REGION Network 158: Lệnh chạy động cơ khuấy Bồn 4 (Coil thường)
   RUNG wire#powerrail
      Contact( "AGTR3263_Should_Run" )
      I_Contact( "PLC2_Loi_Tong" )
      Coil( "AGTR3263_Khuay_Bon4" )
   END_RUNG
   // the same network as SCL:
   "AGTR3263_Khuay_Bon4" := "AGTR3263_Should_Run" AND NOT "PLC2_Loi_Tong";
END_REGION

REGION Network 159: Lệnh đảo chiều động cơ khuấy Bồn 4 (Coil thường)
   RUNG wire#powerrail
      Contact( "PLC2_Step_Bon4_Khuay_Nghich" )
      I_Contact( "PLC2_Loi_Tong" )
      Coil( "AGTR3263_Dao_Chieu" )
   END_RUNG
   // the same network as SCL:
   "AGTR3263_Dao_Chieu" := "PLC2_Step_Bon4_Khuay_Nghich" AND NOT "PLC2_Loi_Tong";
END_REGION

REGION Network 160: Mở van xả đáy Bồn 4 số 1 khi bơm chuyển Nhánh 2 chạy
   RUNG wire#powerrail
      Contact( "Pump3265_Chuyen_Nhanh2" )
      I_Contact( "PLC2_Loi_Tong" )
      Coil( "V3247_Xa_Bon4" )
   END_RUNG
   // the same network as SCL:
   "V3247_Xa_Bon4" := "Pump3265_Chuyen_Nhanh2" AND NOT "PLC2_Loi_Tong";
END_REGION

REGION Network 161: Mở van xả đáy Bồn 4 số 2 khi bơm chuyển Nhánh 2 chạy
   RUNG wire#powerrail
      Contact( "Pump3265_Chuyen_Nhanh2" )
      I_Contact( "PLC2_Loi_Tong" )
      Coil( "V3248_Xa_Bon4" )
   END_RUNG
   // the same network as SCL:
   "V3248_Xa_Bon4" := "Pump3265_Chuyen_Nhanh2" AND NOT "PLC2_Loi_Tong";
END_REGION

REGION Network 162: Mở van xả đáy Bồn 4 số 3 khi bơm chuyển Nhánh 2 chạy
   RUNG wire#powerrail
      Contact( "Pump3265_Chuyen_Nhanh2" )
      I_Contact( "PLC2_Loi_Tong" )
      Coil( "V3249_Xa_Bon4" )
   END_RUNG
   // the same network as SCL:
   "V3249_Xa_Bon4" := "Pump3265_Chuyen_Nhanh2" AND NOT "PLC2_Loi_Tong";
END_REGION

REGION Network 163: Reset CV nước Bồn 3 khi không dosing
   RUNG wire#powerrail
      I_Contact( "PLC2_Step_Bon3_Dosing" )
      { S7_GenerateENO := "TRUE" } Move(in := 0.0, out1 => "CV3211_Nuoc_Bon3")
   END_RUNG
   // the same network as SCL:
   IF NOT "PLC2_Step_Bon3_Dosing" THEN "CV3211_Nuoc_Bon3" := 0.0; END_IF;
END_REGION

REGION Network 164: Reset CV nước Bồn 3 khi Stop hoặc Lỗi tổng PLC2
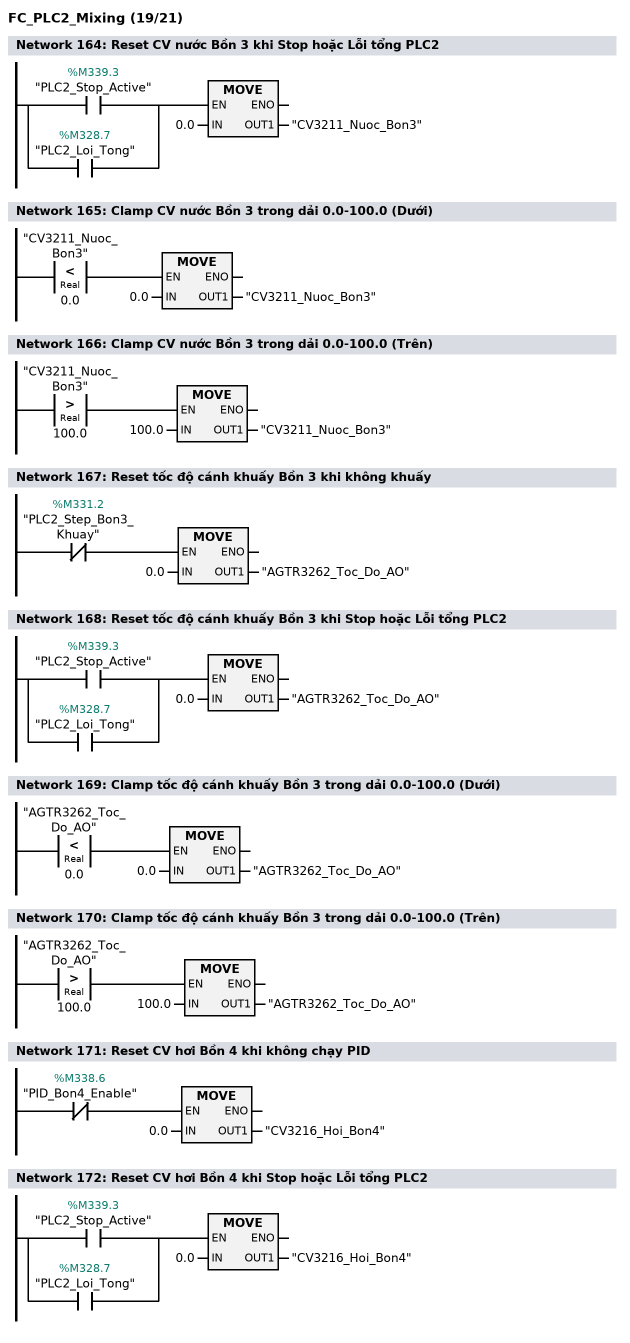
   RUNG wire#powerrail
      Contact( "PLC2_Stop_Active" )
      wire#w1
      { S7_GenerateENO := "TRUE" } Move(in := 0.0, out1 => "CV3211_Nuoc_Bon3")
   END_RUNG
   RUNG wire#powerrail
      Contact( "PLC2_Loi_Tong" )
   END_RUNG wire#w1
   // the same network as SCL:
   IF "PLC2_Stop_Active" OR "PLC2_Loi_Tong" THEN "CV3211_Nuoc_Bon3" := 0.0; END_IF;
END_REGION

REGION Network 165: Clamp CV nước Bồn 3 trong dải 0.0-100.0 (Dưới)
   RUNG wire#powerrail
      { S7_Templates := "SrcType := Real" } LT_Contact(in1 := "CV3211_Nuoc_Bon3", in2 := 0.0)
      { S7_GenerateENO := "TRUE" } Move(in := 0.0, out1 => "CV3211_Nuoc_Bon3")
   END_RUNG
   // the same network as SCL:
   IF "CV3211_Nuoc_Bon3" < 0.0 THEN "CV3211_Nuoc_Bon3" := 0.0; END_IF;
END_REGION

REGION Network 166: Clamp CV nước Bồn 3 trong dải 0.0-100.0 (Trên)
   RUNG wire#powerrail
      { S7_Templates := "SrcType := Real" } GT_Contact(in1 := "CV3211_Nuoc_Bon3", in2 := 100.0)
      { S7_GenerateENO := "TRUE" } Move(in := 100.0, out1 => "CV3211_Nuoc_Bon3")
   END_RUNG
   // the same network as SCL:
   IF "CV3211_Nuoc_Bon3" > 100.0 THEN "CV3211_Nuoc_Bon3" := 100.0; END_IF;
END_REGION

REGION Network 167: Reset tốc độ cánh khuấy Bồn 3 khi không khuấy
   RUNG wire#powerrail
      I_Contact( "PLC2_Step_Bon3_Khuay" )
      { S7_GenerateENO := "TRUE" } Move(in := 0.0, out1 => "AGTR3262_Toc_Do_AO")
   END_RUNG
   // the same network as SCL:
   IF NOT "PLC2_Step_Bon3_Khuay" THEN "AGTR3262_Toc_Do_AO" := 0.0; END_IF;
END_REGION

REGION Network 168: Reset tốc độ cánh khuấy Bồn 3 khi Stop hoặc Lỗi tổng PLC2
   RUNG wire#powerrail
      Contact( "PLC2_Stop_Active" )
      wire#w1
      { S7_GenerateENO := "TRUE" } Move(in := 0.0, out1 => "AGTR3262_Toc_Do_AO")
   END_RUNG
   RUNG wire#powerrail
      Contact( "PLC2_Loi_Tong" )
   END_RUNG wire#w1
   // the same network as SCL:
   IF "PLC2_Stop_Active" OR "PLC2_Loi_Tong" THEN "AGTR3262_Toc_Do_AO" := 0.0; END_IF;
END_REGION

REGION Network 169: Clamp tốc độ cánh khuấy Bồn 3 trong dải 0.0-100.0 (Dưới)
   RUNG wire#powerrail
      { S7_Templates := "SrcType := Real" } LT_Contact(in1 := "AGTR3262_Toc_Do_AO", in2 := 0.0)
      { S7_GenerateENO := "TRUE" } Move(in := 0.0, out1 => "AGTR3262_Toc_Do_AO")
   END_RUNG
   // the same network as SCL:
   IF "AGTR3262_Toc_Do_AO" < 0.0 THEN "AGTR3262_Toc_Do_AO" := 0.0; END_IF;
END_REGION

REGION Network 170: Clamp tốc độ cánh khuấy Bồn 3 trong dải 0.0-100.0 (Trên)
   RUNG wire#powerrail
      { S7_Templates := "SrcType := Real" } GT_Contact(in1 := "AGTR3262_Toc_Do_AO", in2 := 100.0)
      { S7_GenerateENO := "TRUE" } Move(in := 100.0, out1 => "AGTR3262_Toc_Do_AO")
   END_RUNG
   // the same network as SCL:
   IF "AGTR3262_Toc_Do_AO" > 100.0 THEN "AGTR3262_Toc_Do_AO" := 100.0; END_IF;
END_REGION

REGION Network 171: Reset CV hơi Bồn 4 khi không chạy PID
   RUNG wire#powerrail
      I_Contact( "PID_Bon4_Enable" )
      { S7_GenerateENO := "TRUE" } Move(in := 0.0, out1 => "CV3216_Hoi_Bon4")
   END_RUNG
   // the same network as SCL:
   IF NOT "PID_Bon4_Enable" THEN "CV3216_Hoi_Bon4" := 0.0; END_IF;
END_REGION

REGION Network 172: Reset CV hơi Bồn 4 khi Stop hoặc Lỗi tổng PLC2
   RUNG wire#powerrail
      Contact( "PLC2_Stop_Active" )
      wire#w1
      { S7_GenerateENO := "TRUE" } Move(in := 0.0, out1 => "CV3216_Hoi_Bon4")
   END_RUNG
   RUNG wire#powerrail
      Contact( "PLC2_Loi_Tong" )
   END_RUNG wire#w1
   // the same network as SCL:
   IF "PLC2_Stop_Active" OR "PLC2_Loi_Tong" THEN "CV3216_Hoi_Bon4" := 0.0; END_IF;
END_REGION

REGION Network 173: Clamp CV hơi Bồn 4 trong dải 0.0-100.0 (Dưới)
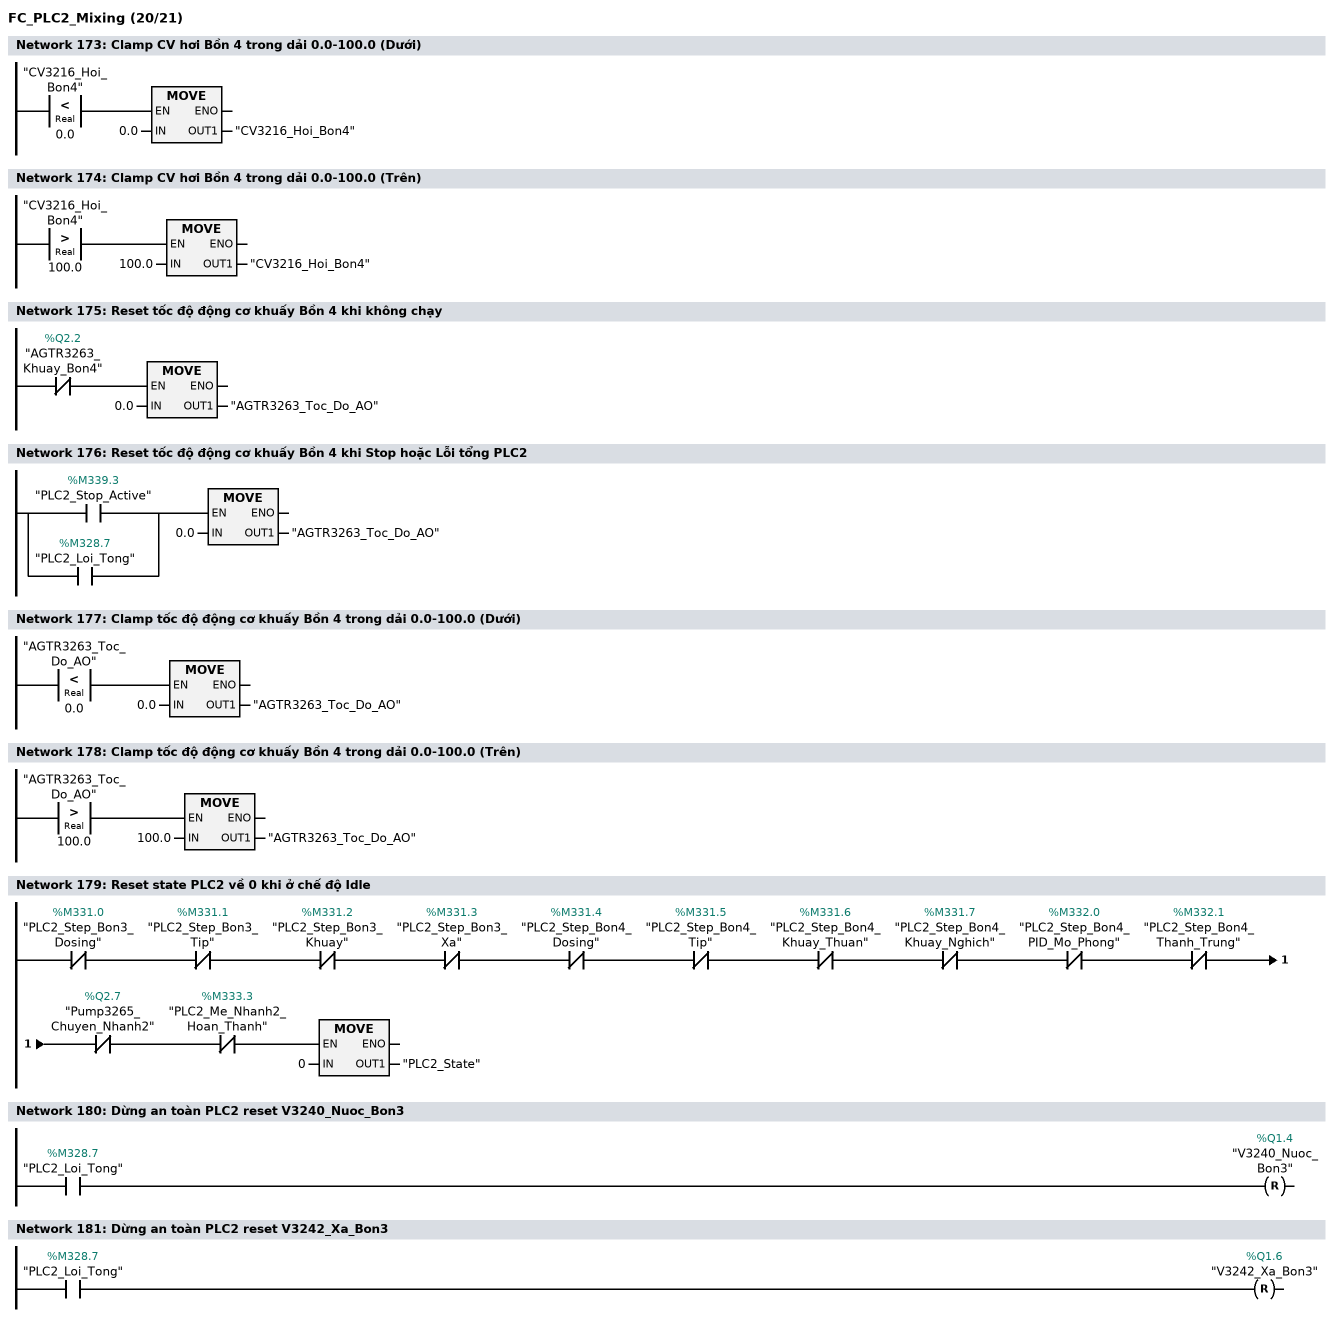
   RUNG wire#powerrail
      { S7_Templates := "SrcType := Real" } LT_Contact(in1 := "CV3216_Hoi_Bon4", in2 := 0.0)
      { S7_GenerateENO := "TRUE" } Move(in := 0.0, out1 => "CV3216_Hoi_Bon4")
   END_RUNG
   // the same network as SCL:
   IF "CV3216_Hoi_Bon4" < 0.0 THEN "CV3216_Hoi_Bon4" := 0.0; END_IF;
END_REGION

REGION Network 174: Clamp CV hơi Bồn 4 trong dải 0.0-100.0 (Trên)
   RUNG wire#powerrail
      { S7_Templates := "SrcType := Real" } GT_Contact(in1 := "CV3216_Hoi_Bon4", in2 := 100.0)
      { S7_GenerateENO := "TRUE" } Move(in := 100.0, out1 => "CV3216_Hoi_Bon4")
   END_RUNG
   // the same network as SCL:
   IF "CV3216_Hoi_Bon4" > 100.0 THEN "CV3216_Hoi_Bon4" := 100.0; END_IF;
END_REGION

REGION Network 175: Reset tốc độ động cơ khuấy Bồn 4 khi không chạy
   RUNG wire#powerrail
      I_Contact( "AGTR3263_Khuay_Bon4" )
      { S7_GenerateENO := "TRUE" } Move(in := 0.0, out1 => "AGTR3263_Toc_Do_AO")
   END_RUNG
   // the same network as SCL:
   IF NOT "AGTR3263_Khuay_Bon4" THEN "AGTR3263_Toc_Do_AO" := 0.0; END_IF;
END_REGION

REGION Network 176: Reset tốc độ động cơ khuấy Bồn 4 khi Stop hoặc Lỗi tổng PLC2
   RUNG wire#powerrail
      Contact( "PLC2_Stop_Active" )
      wire#w1
      { S7_GenerateENO := "TRUE" } Move(in := 0.0, out1 => "AGTR3263_Toc_Do_AO")
   END_RUNG
   RUNG wire#powerrail
      Contact( "PLC2_Loi_Tong" )
   END_RUNG wire#w1
   // the same network as SCL:
   IF "PLC2_Stop_Active" OR "PLC2_Loi_Tong" THEN "AGTR3263_Toc_Do_AO" := 0.0; END_IF;
END_REGION

REGION Network 177: Clamp tốc độ động cơ khuấy Bồn 4 trong dải 0.0-100.0 (Dưới)
   RUNG wire#powerrail
      { S7_Templates := "SrcType := Real" } LT_Contact(in1 := "AGTR3263_Toc_Do_AO", in2 := 0.0)
      { S7_GenerateENO := "TRUE" } Move(in := 0.0, out1 => "AGTR3263_Toc_Do_AO")
   END_RUNG
   // the same network as SCL:
   IF "AGTR3263_Toc_Do_AO" < 0.0 THEN "AGTR3263_Toc_Do_AO" := 0.0; END_IF;
END_REGION

REGION Network 178: Clamp tốc độ động cơ khuấy Bồn 4 trong dải 0.0-100.0 (Trên)
   RUNG wire#powerrail
      { S7_Templates := "SrcType := Real" } GT_Contact(in1 := "AGTR3263_Toc_Do_AO", in2 := 100.0)
      { S7_GenerateENO := "TRUE" } Move(in := 100.0, out1 => "AGTR3263_Toc_Do_AO")
   END_RUNG
   // the same network as SCL:
   IF "AGTR3263_Toc_Do_AO" > 100.0 THEN "AGTR3263_Toc_Do_AO" := 100.0; END_IF;
END_REGION

REGION Network 179: Reset state PLC2 về 0 khi ở chế độ Idle
   RUNG wire#powerrail
      I_Contact( "PLC2_Step_Bon3_Dosing" )
      I_Contact( "PLC2_Step_Bon3_Tip" )
      I_Contact( "PLC2_Step_Bon3_Khuay" )
      I_Contact( "PLC2_Step_Bon3_Xa" )
      I_Contact( "PLC2_Step_Bon4_Dosing" )
      I_Contact( "PLC2_Step_Bon4_Tip" )
      I_Contact( "PLC2_Step_Bon4_Khuay_Thuan" )
      I_Contact( "PLC2_Step_Bon4_Khuay_Nghich" )
      I_Contact( "PLC2_Step_Bon4_PID_Mo_Phong" )
      I_Contact( "PLC2_Step_Bon4_Thanh_Trung" )
      I_Contact( "Pump3265_Chuyen_Nhanh2" )
      I_Contact( "PLC2_Me_Nhanh2_Hoan_Thanh" )
      { S7_GenerateENO := "TRUE" } Move(in := 0, out1 => "PLC2_State")
   END_RUNG
   // the same network as SCL:
   IF NOT "PLC2_Step_Bon3_Dosing" AND NOT "PLC2_Step_Bon3_Tip" AND NOT "PLC2_Step_Bon3_Khuay" AND NOT "PLC2_Step_Bon3_Xa" AND NOT "PLC2_Step_Bon4_Dosing" AND NOT "PLC2_Step_Bon4_Tip" AND NOT "PLC2_Step_Bon4_Khuay_Thuan" AND NOT "PLC2_Step_Bon4_Khuay_Nghich" AND NOT "PLC2_Step_Bon4_PID_Mo_Phong" AND NOT "PLC2_Step_Bon4_Thanh_Trung" AND NOT "Pump3265_Chuyen_Nhanh2" AND NOT "PLC2_Me_Nhanh2_Hoan_Thanh" THEN
       "PLC2_State" := 0;
   END_IF;
END_REGION

REGION Network 180: Dừng an toàn PLC2 reset V3240_Nuoc_Bon3
   RUNG wire#powerrail
      Contact( "PLC2_Loi_Tong" )
      R_Coil( "V3240_Nuoc_Bon3" )
   END_RUNG
   // the same network as SCL:
   IF "PLC2_Loi_Tong" THEN "V3240_Nuoc_Bon3" := FALSE; END_IF;
END_REGION

REGION Network 181: Dừng an toàn PLC2 reset V3242_Xa_Bon3
   RUNG wire#powerrail
      Contact( "PLC2_Loi_Tong" )
      R_Coil( "V3242_Xa_Bon3" )
   END_RUNG
   // the same network as SCL:
   IF "PLC2_Loi_Tong" THEN "V3242_Xa_Bon3" := FALSE; END_IF;
END_REGION

REGION Network 182: Dừng an toàn PLC2 reset V3243_Xa_Bon3
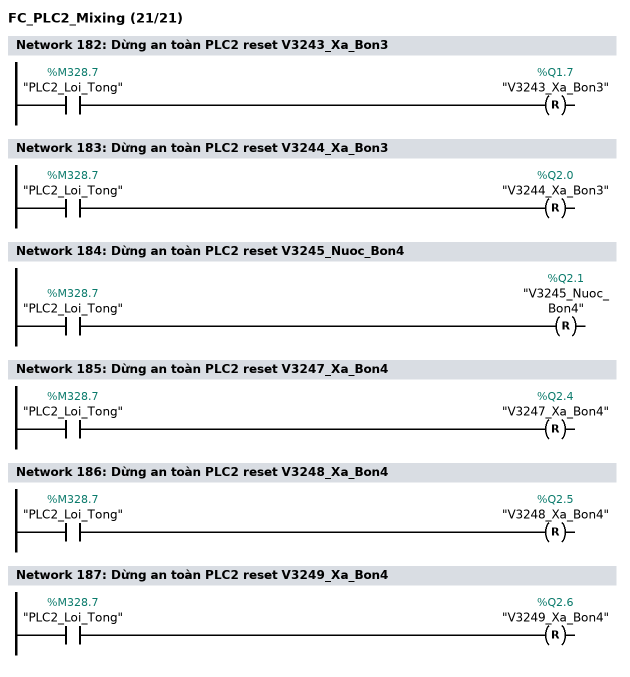
   RUNG wire#powerrail
      Contact( "PLC2_Loi_Tong" )
      R_Coil( "V3243_Xa_Bon3" )
   END_RUNG
   // the same network as SCL:
   IF "PLC2_Loi_Tong" THEN "V3243_Xa_Bon3" := FALSE; END_IF;
END_REGION

REGION Network 183: Dừng an toàn PLC2 reset V3244_Xa_Bon3
   RUNG wire#powerrail
      Contact( "PLC2_Loi_Tong" )
      R_Coil( "V3244_Xa_Bon3" )
   END_RUNG
   // the same network as SCL:
   IF "PLC2_Loi_Tong" THEN "V3244_Xa_Bon3" := FALSE; END_IF;
END_REGION

REGION Network 184: Dừng an toàn PLC2 reset V3245_Nuoc_Bon4
   RUNG wire#powerrail
      Contact( "PLC2_Loi_Tong" )
      R_Coil( "V3245_Nuoc_Bon4" )
   END_RUNG
   // the same network as SCL:
   IF "PLC2_Loi_Tong" THEN "V3245_Nuoc_Bon4" := FALSE; END_IF;
END_REGION

REGION Network 185: Dừng an toàn PLC2 reset V3247_Xa_Bon4
   RUNG wire#powerrail
      Contact( "PLC2_Loi_Tong" )
      R_Coil( "V3247_Xa_Bon4" )
   END_RUNG
   // the same network as SCL:
   IF "PLC2_Loi_Tong" THEN "V3247_Xa_Bon4" := FALSE; END_IF;
END_REGION

REGION Network 186: Dừng an toàn PLC2 reset V3248_Xa_Bon4
   RUNG wire#powerrail
      Contact( "PLC2_Loi_Tong" )
      R_Coil( "V3248_Xa_Bon4" )
   END_RUNG
   // the same network as SCL:
   IF "PLC2_Loi_Tong" THEN "V3248_Xa_Bon4" := FALSE; END_IF;
END_REGION

REGION Network 187: Dừng an toàn PLC2 reset V3249_Xa_Bon4
   RUNG wire#powerrail
      Contact( "PLC2_Loi_Tong" )
      R_Coil( "V3249_Xa_Bon4" )
   END_RUNG
   // the same network as SCL:
   IF "PLC2_Loi_Tong" THEN "V3249_Xa_Bon4" := FALSE; END_IF;
END_REGION
END_FUNCTION

FUNCTION "FC_Manual_Control_PLC2" : Void   // FC62, LAD
{ S7_Optimized_Access := 'TRUE' }
VERSION : 0.1
// stored: AutoNumber true, IsIECCheckEnabled false, SetENOAutomatically false, UDAEnableTagReadback false
BEGIN

REGION Network 1: Xác định trạng thái Manual Mode Active PLC2
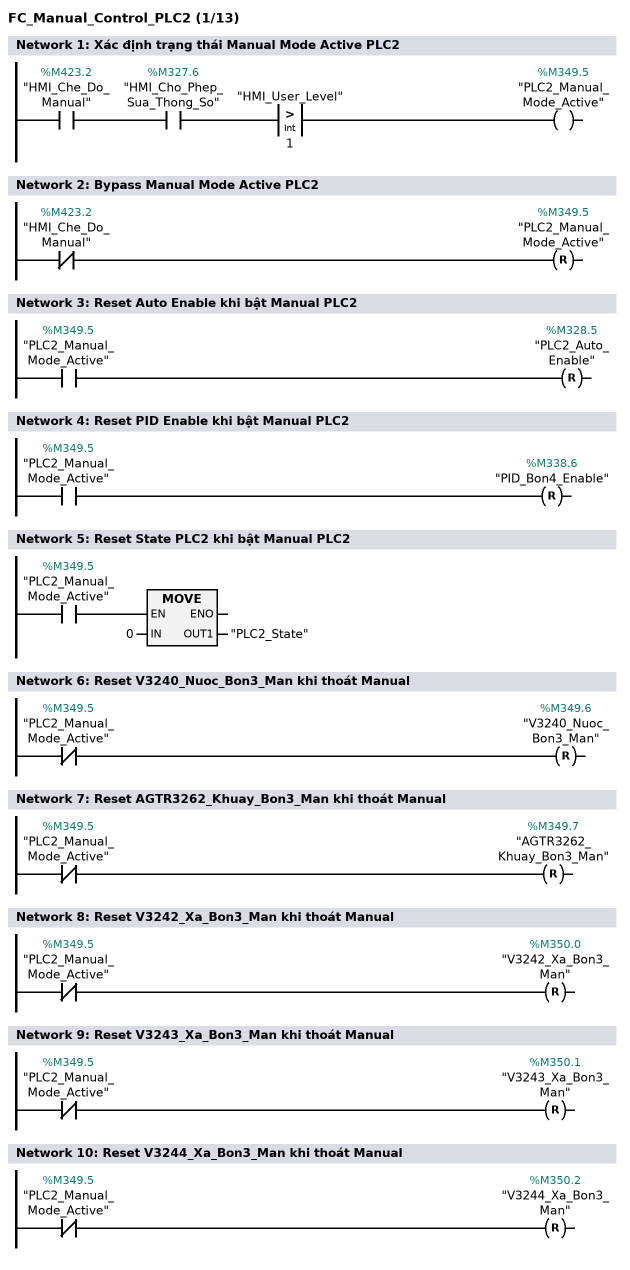
   RUNG wire#powerrail
      Contact( "HMI_Che_Do_Manual" )
      Contact( "HMI_Cho_Phep_Sua_Thong_So" )
      { S7_Templates := "SrcType := Int" } GT_Contact(in1 := "HMI_User_Level", in2 := 1)
      Coil( "PLC2_Manual_Mode_Active" )
   END_RUNG
   // the same network as SCL:
   "PLC2_Manual_Mode_Active" := "HMI_Che_Do_Manual" AND "HMI_Cho_Phep_Sua_Thong_So" AND ("HMI_User_Level" > 1);
END_REGION

REGION Network 2: Bypass Manual Mode Active PLC2
   RUNG wire#powerrail
      I_Contact( "HMI_Che_Do_Manual" )
      R_Coil( "PLC2_Manual_Mode_Active" )
   END_RUNG
   // the same network as SCL:
   IF NOT "HMI_Che_Do_Manual" THEN "PLC2_Manual_Mode_Active" := FALSE; END_IF;
END_REGION

REGION Network 3: Reset Auto Enable khi bật Manual PLC2
   RUNG wire#powerrail
      Contact( "PLC2_Manual_Mode_Active" )
      R_Coil( "PLC2_Auto_Enable" )
   END_RUNG
   // the same network as SCL:
   IF "PLC2_Manual_Mode_Active" THEN "PLC2_Auto_Enable" := FALSE; END_IF;
END_REGION

REGION Network 4: Reset PID Enable khi bật Manual PLC2
   RUNG wire#powerrail
      Contact( "PLC2_Manual_Mode_Active" )
      R_Coil( "PID_Bon4_Enable" )
   END_RUNG
   // the same network as SCL:
   IF "PLC2_Manual_Mode_Active" THEN "PID_Bon4_Enable" := FALSE; END_IF;
END_REGION

REGION Network 5: Reset State PLC2 khi bật Manual PLC2
   RUNG wire#powerrail
      Contact( "PLC2_Manual_Mode_Active" )
      { S7_GenerateENO := "TRUE" } Move(in := 0, out1 => "PLC2_State")
   END_RUNG
   // the same network as SCL:
   IF "PLC2_Manual_Mode_Active" THEN "PLC2_State" := 0; END_IF;
END_REGION

REGION Network 6: Reset V3240_Nuoc_Bon3_Man khi thoát Manual
   RUNG wire#powerrail
      I_Contact( "PLC2_Manual_Mode_Active" )
      R_Coil( "V3240_Nuoc_Bon3_Man" )
   END_RUNG
   // the same network as SCL:
   IF NOT "PLC2_Manual_Mode_Active" THEN "V3240_Nuoc_Bon3_Man" := FALSE; END_IF;
END_REGION

REGION Network 7: Reset AGTR3262_Khuay_Bon3_Man khi thoát Manual
   RUNG wire#powerrail
      I_Contact( "PLC2_Manual_Mode_Active" )
      R_Coil( "AGTR3262_Khuay_Bon3_Man" )
   END_RUNG
   // the same network as SCL:
   IF NOT "PLC2_Manual_Mode_Active" THEN "AGTR3262_Khuay_Bon3_Man" := FALSE; END_IF;
END_REGION

REGION Network 8: Reset V3242_Xa_Bon3_Man khi thoát Manual
   RUNG wire#powerrail
      I_Contact( "PLC2_Manual_Mode_Active" )
      R_Coil( "V3242_Xa_Bon3_Man" )
   END_RUNG
   // the same network as SCL:
   IF NOT "PLC2_Manual_Mode_Active" THEN "V3242_Xa_Bon3_Man" := FALSE; END_IF;
END_REGION

REGION Network 9: Reset V3243_Xa_Bon3_Man khi thoát Manual
   RUNG wire#powerrail
      I_Contact( "PLC2_Manual_Mode_Active" )
      R_Coil( "V3243_Xa_Bon3_Man" )
   END_RUNG
   // the same network as SCL:
   IF NOT "PLC2_Manual_Mode_Active" THEN "V3243_Xa_Bon3_Man" := FALSE; END_IF;
END_REGION

REGION Network 10: Reset V3244_Xa_Bon3_Man khi thoát Manual
   RUNG wire#powerrail
      I_Contact( "PLC2_Manual_Mode_Active" )
      R_Coil( "V3244_Xa_Bon3_Man" )
   END_RUNG
   // the same network as SCL:
   IF NOT "PLC2_Manual_Mode_Active" THEN "V3244_Xa_Bon3_Man" := FALSE; END_IF;
END_REGION

REGION Network 11: Reset V3245_Nuoc_Bon4_Man khi thoát Manual
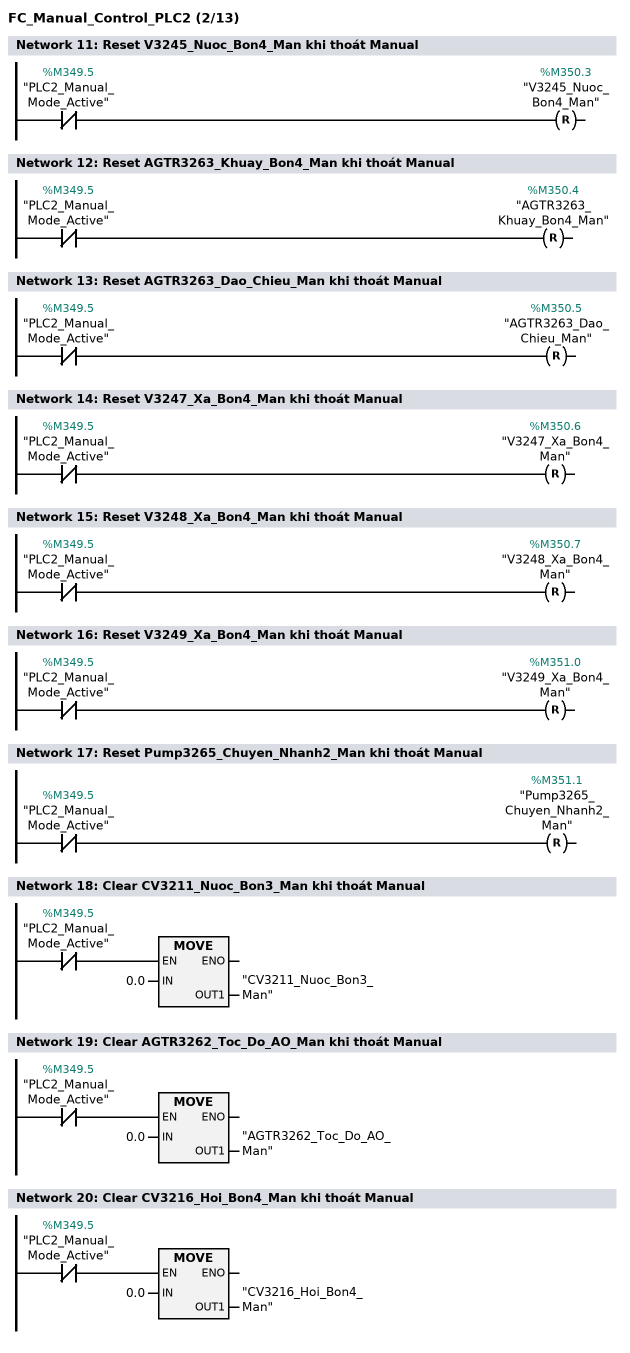
   RUNG wire#powerrail
      I_Contact( "PLC2_Manual_Mode_Active" )
      R_Coil( "V3245_Nuoc_Bon4_Man" )
   END_RUNG
   // the same network as SCL:
   IF NOT "PLC2_Manual_Mode_Active" THEN "V3245_Nuoc_Bon4_Man" := FALSE; END_IF;
END_REGION

REGION Network 12: Reset AGTR3263_Khuay_Bon4_Man khi thoát Manual
   RUNG wire#powerrail
      I_Contact( "PLC2_Manual_Mode_Active" )
      R_Coil( "AGTR3263_Khuay_Bon4_Man" )
   END_RUNG
   // the same network as SCL:
   IF NOT "PLC2_Manual_Mode_Active" THEN "AGTR3263_Khuay_Bon4_Man" := FALSE; END_IF;
END_REGION

REGION Network 13: Reset AGTR3263_Dao_Chieu_Man khi thoát Manual
   RUNG wire#powerrail
      I_Contact( "PLC2_Manual_Mode_Active" )
      R_Coil( "AGTR3263_Dao_Chieu_Man" )
   END_RUNG
   // the same network as SCL:
   IF NOT "PLC2_Manual_Mode_Active" THEN "AGTR3263_Dao_Chieu_Man" := FALSE; END_IF;
END_REGION

REGION Network 14: Reset V3247_Xa_Bon4_Man khi thoát Manual
   RUNG wire#powerrail
      I_Contact( "PLC2_Manual_Mode_Active" )
      R_Coil( "V3247_Xa_Bon4_Man" )
   END_RUNG
   // the same network as SCL:
   IF NOT "PLC2_Manual_Mode_Active" THEN "V3247_Xa_Bon4_Man" := FALSE; END_IF;
END_REGION

REGION Network 15: Reset V3248_Xa_Bon4_Man khi thoát Manual
   RUNG wire#powerrail
      I_Contact( "PLC2_Manual_Mode_Active" )
      R_Coil( "V3248_Xa_Bon4_Man" )
   END_RUNG
   // the same network as SCL:
   IF NOT "PLC2_Manual_Mode_Active" THEN "V3248_Xa_Bon4_Man" := FALSE; END_IF;
END_REGION

REGION Network 16: Reset V3249_Xa_Bon4_Man khi thoát Manual
   RUNG wire#powerrail
      I_Contact( "PLC2_Manual_Mode_Active" )
      R_Coil( "V3249_Xa_Bon4_Man" )
   END_RUNG
   // the same network as SCL:
   IF NOT "PLC2_Manual_Mode_Active" THEN "V3249_Xa_Bon4_Man" := FALSE; END_IF;
END_REGION

REGION Network 17: Reset Pump3265_Chuyen_Nhanh2_Man khi thoát Manual
   RUNG wire#powerrail
      I_Contact( "PLC2_Manual_Mode_Active" )
      R_Coil( "Pump3265_Chuyen_Nhanh2_Man" )
   END_RUNG
   // the same network as SCL:
   IF NOT "PLC2_Manual_Mode_Active" THEN "Pump3265_Chuyen_Nhanh2_Man" := FALSE; END_IF;
END_REGION

REGION Network 18: Clear CV3211_Nuoc_Bon3_Man khi thoát Manual
   RUNG wire#powerrail
      I_Contact( "PLC2_Manual_Mode_Active" )
      { S7_GenerateENO := "TRUE" } Move(in := 0.0, out1 => "CV3211_Nuoc_Bon3_Man")
   END_RUNG
   // the same network as SCL:
   IF NOT "PLC2_Manual_Mode_Active" THEN "CV3211_Nuoc_Bon3_Man" := 0.0; END_IF;
END_REGION

REGION Network 19: Clear AGTR3262_Toc_Do_AO_Man khi thoát Manual
   RUNG wire#powerrail
      I_Contact( "PLC2_Manual_Mode_Active" )
      { S7_GenerateENO := "TRUE" } Move(in := 0.0, out1 => "AGTR3262_Toc_Do_AO_Man")
   END_RUNG
   // the same network as SCL:
   IF NOT "PLC2_Manual_Mode_Active" THEN "AGTR3262_Toc_Do_AO_Man" := 0.0; END_IF;
END_REGION

REGION Network 20: Clear CV3216_Hoi_Bon4_Man khi thoát Manual
   RUNG wire#powerrail
      I_Contact( "PLC2_Manual_Mode_Active" )
      { S7_GenerateENO := "TRUE" } Move(in := 0.0, out1 => "CV3216_Hoi_Bon4_Man")
   END_RUNG
   // the same network as SCL:
   IF NOT "PLC2_Manual_Mode_Active" THEN "CV3216_Hoi_Bon4_Man" := 0.0; END_IF;
END_REGION

REGION Network 21: Clear AGTR3263_Toc_Do_AO_Man khi thoát Manual
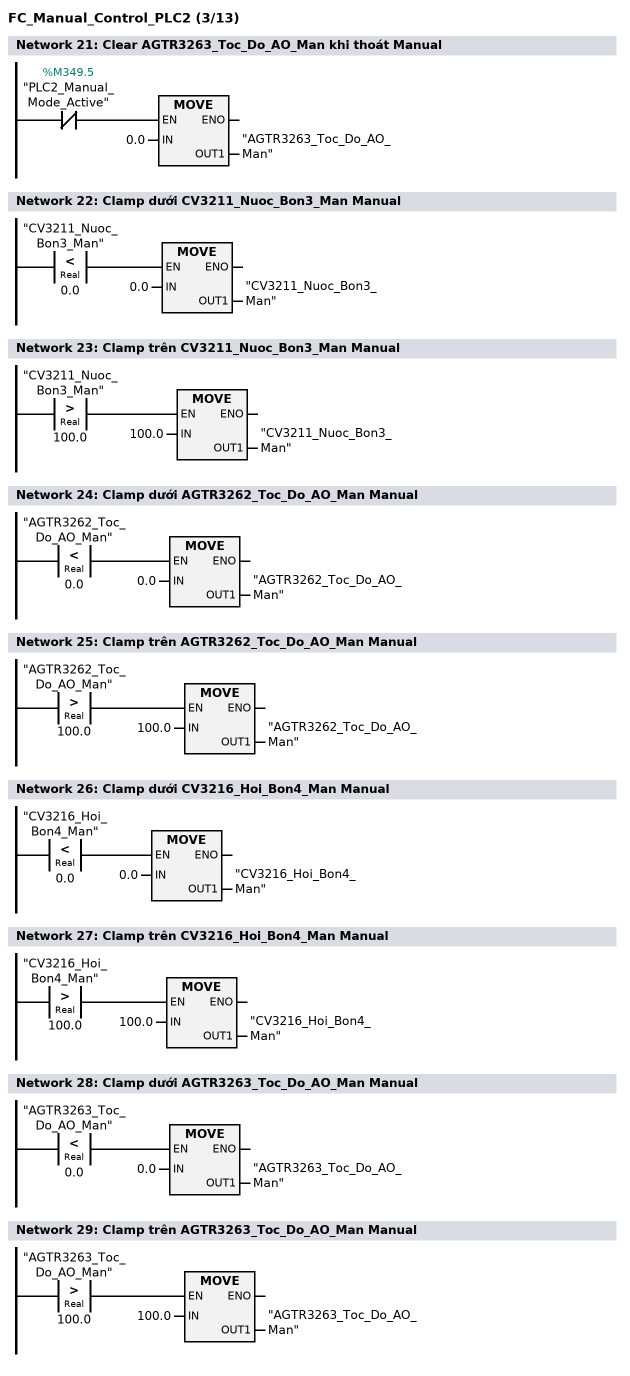
   RUNG wire#powerrail
      I_Contact( "PLC2_Manual_Mode_Active" )
      { S7_GenerateENO := "TRUE" } Move(in := 0.0, out1 => "AGTR3263_Toc_Do_AO_Man")
   END_RUNG
   // the same network as SCL:
   IF NOT "PLC2_Manual_Mode_Active" THEN "AGTR3263_Toc_Do_AO_Man" := 0.0; END_IF;
END_REGION

REGION Network 22: Clamp dưới CV3211_Nuoc_Bon3_Man Manual
   RUNG wire#powerrail
      { S7_Templates := "SrcType := Real" } LT_Contact(in1 := "CV3211_Nuoc_Bon3_Man", in2 := 0.0)
      { S7_GenerateENO := "TRUE" } Move(in := 0.0, out1 => "CV3211_Nuoc_Bon3_Man")
   END_RUNG
   // the same network as SCL:
   IF "CV3211_Nuoc_Bon3_Man" < 0.0 THEN "CV3211_Nuoc_Bon3_Man" := 0.0; END_IF;
END_REGION

REGION Network 23: Clamp trên CV3211_Nuoc_Bon3_Man Manual
   RUNG wire#powerrail
      { S7_Templates := "SrcType := Real" } GT_Contact(in1 := "CV3211_Nuoc_Bon3_Man", in2 := 100.0)
      { S7_GenerateENO := "TRUE" } Move(in := 100.0, out1 => "CV3211_Nuoc_Bon3_Man")
   END_RUNG
   // the same network as SCL:
   IF "CV3211_Nuoc_Bon3_Man" > 100.0 THEN "CV3211_Nuoc_Bon3_Man" := 100.0; END_IF;
END_REGION

REGION Network 24: Clamp dưới AGTR3262_Toc_Do_AO_Man Manual
   RUNG wire#powerrail
      { S7_Templates := "SrcType := Real" } LT_Contact(in1 := "AGTR3262_Toc_Do_AO_Man", in2 := 0.0)
      { S7_GenerateENO := "TRUE" } Move(in := 0.0, out1 => "AGTR3262_Toc_Do_AO_Man")
   END_RUNG
   // the same network as SCL:
   IF "AGTR3262_Toc_Do_AO_Man" < 0.0 THEN "AGTR3262_Toc_Do_AO_Man" := 0.0; END_IF;
END_REGION

REGION Network 25: Clamp trên AGTR3262_Toc_Do_AO_Man Manual
   RUNG wire#powerrail
      { S7_Templates := "SrcType := Real" } GT_Contact(in1 := "AGTR3262_Toc_Do_AO_Man", in2 := 100.0)
      { S7_GenerateENO := "TRUE" } Move(in := 100.0, out1 => "AGTR3262_Toc_Do_AO_Man")
   END_RUNG
   // the same network as SCL:
   IF "AGTR3262_Toc_Do_AO_Man" > 100.0 THEN "AGTR3262_Toc_Do_AO_Man" := 100.0; END_IF;
END_REGION

REGION Network 26: Clamp dưới CV3216_Hoi_Bon4_Man Manual
   RUNG wire#powerrail
      { S7_Templates := "SrcType := Real" } LT_Contact(in1 := "CV3216_Hoi_Bon4_Man", in2 := 0.0)
      { S7_GenerateENO := "TRUE" } Move(in := 0.0, out1 => "CV3216_Hoi_Bon4_Man")
   END_RUNG
   // the same network as SCL:
   IF "CV3216_Hoi_Bon4_Man" < 0.0 THEN "CV3216_Hoi_Bon4_Man" := 0.0; END_IF;
END_REGION

REGION Network 27: Clamp trên CV3216_Hoi_Bon4_Man Manual
   RUNG wire#powerrail
      { S7_Templates := "SrcType := Real" } GT_Contact(in1 := "CV3216_Hoi_Bon4_Man", in2 := 100.0)
      { S7_GenerateENO := "TRUE" } Move(in := 100.0, out1 => "CV3216_Hoi_Bon4_Man")
   END_RUNG
   // the same network as SCL:
   IF "CV3216_Hoi_Bon4_Man" > 100.0 THEN "CV3216_Hoi_Bon4_Man" := 100.0; END_IF;
END_REGION

REGION Network 28: Clamp dưới AGTR3263_Toc_Do_AO_Man Manual
   RUNG wire#powerrail
      { S7_Templates := "SrcType := Real" } LT_Contact(in1 := "AGTR3263_Toc_Do_AO_Man", in2 := 0.0)
      { S7_GenerateENO := "TRUE" } Move(in := 0.0, out1 => "AGTR3263_Toc_Do_AO_Man")
   END_RUNG
   // the same network as SCL:
   IF "AGTR3263_Toc_Do_AO_Man" < 0.0 THEN "AGTR3263_Toc_Do_AO_Man" := 0.0; END_IF;
END_REGION

REGION Network 29: Clamp trên AGTR3263_Toc_Do_AO_Man Manual
   RUNG wire#powerrail
      { S7_Templates := "SrcType := Real" } GT_Contact(in1 := "AGTR3263_Toc_Do_AO_Man", in2 := 100.0)
      { S7_GenerateENO := "TRUE" } Move(in := 100.0, out1 => "AGTR3263_Toc_Do_AO_Man")
   END_RUNG
   // the same network as SCL:
   IF "AGTR3263_Toc_Do_AO_Man" > 100.0 THEN "AGTR3263_Toc_Do_AO_Man" := 100.0; END_IF;
END_REGION

REGION Network 30: Manual V3240_Nuoc_Bon3 - Set
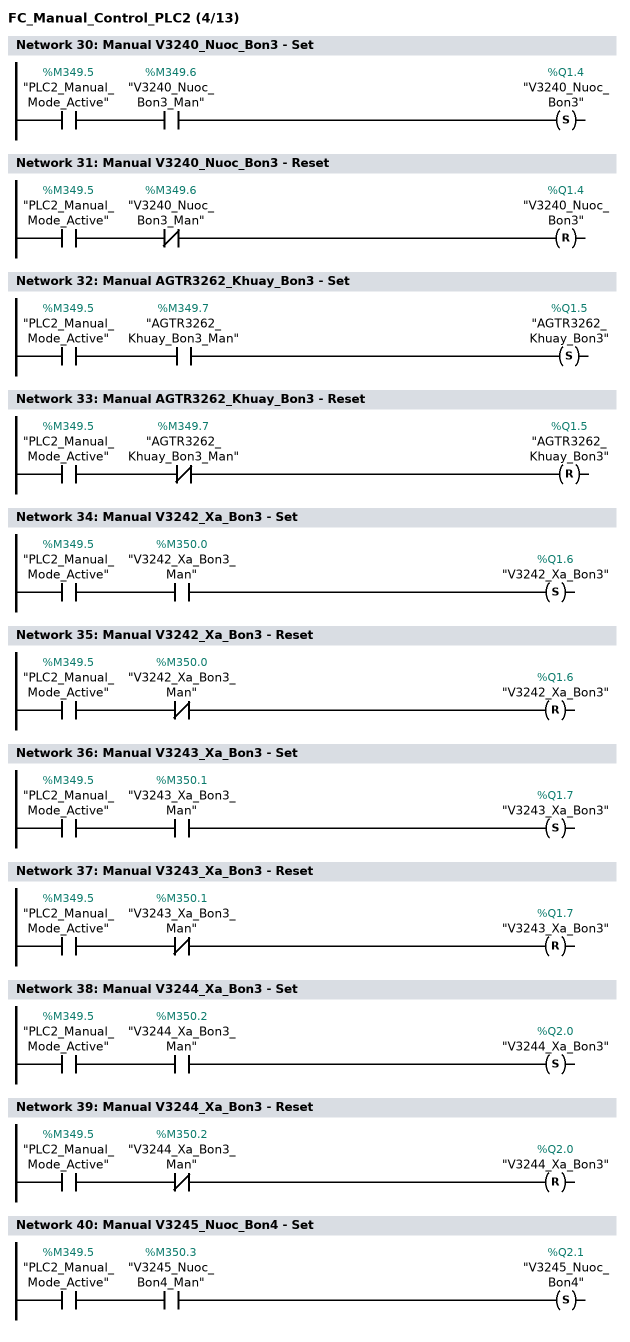
   RUNG wire#powerrail
      Contact( "PLC2_Manual_Mode_Active" )
      Contact( "V3240_Nuoc_Bon3_Man" )
      S_Coil( "V3240_Nuoc_Bon3" )
   END_RUNG
   // the same network as SCL:
   IF "PLC2_Manual_Mode_Active" AND "V3240_Nuoc_Bon3_Man" THEN "V3240_Nuoc_Bon3" := TRUE; END_IF;
END_REGION

REGION Network 31: Manual V3240_Nuoc_Bon3 - Reset
   RUNG wire#powerrail
      Contact( "PLC2_Manual_Mode_Active" )
      I_Contact( "V3240_Nuoc_Bon3_Man" )
      R_Coil( "V3240_Nuoc_Bon3" )
   END_RUNG
   // the same network as SCL:
   IF "PLC2_Manual_Mode_Active" AND NOT "V3240_Nuoc_Bon3_Man" THEN "V3240_Nuoc_Bon3" := FALSE; END_IF;
END_REGION

REGION Network 32: Manual AGTR3262_Khuay_Bon3 - Set
   RUNG wire#powerrail
      Contact( "PLC2_Manual_Mode_Active" )
      Contact( "AGTR3262_Khuay_Bon3_Man" )
      S_Coil( "AGTR3262_Khuay_Bon3" )
   END_RUNG
   // the same network as SCL:
   IF "PLC2_Manual_Mode_Active" AND "AGTR3262_Khuay_Bon3_Man" THEN "AGTR3262_Khuay_Bon3" := TRUE; END_IF;
END_REGION

REGION Network 33: Manual AGTR3262_Khuay_Bon3 - Reset
   RUNG wire#powerrail
      Contact( "PLC2_Manual_Mode_Active" )
      I_Contact( "AGTR3262_Khuay_Bon3_Man" )
      R_Coil( "AGTR3262_Khuay_Bon3" )
   END_RUNG
   // the same network as SCL:
   IF "PLC2_Manual_Mode_Active" AND NOT "AGTR3262_Khuay_Bon3_Man" THEN
       "AGTR3262_Khuay_Bon3" := FALSE;
   END_IF;
END_REGION

REGION Network 34: Manual V3242_Xa_Bon3 - Set
   RUNG wire#powerrail
      Contact( "PLC2_Manual_Mode_Active" )
      Contact( "V3242_Xa_Bon3_Man" )
      S_Coil( "V3242_Xa_Bon3" )
   END_RUNG
   // the same network as SCL:
   IF "PLC2_Manual_Mode_Active" AND "V3242_Xa_Bon3_Man" THEN "V3242_Xa_Bon3" := TRUE; END_IF;
END_REGION

REGION Network 35: Manual V3242_Xa_Bon3 - Reset
   RUNG wire#powerrail
      Contact( "PLC2_Manual_Mode_Active" )
      I_Contact( "V3242_Xa_Bon3_Man" )
      R_Coil( "V3242_Xa_Bon3" )
   END_RUNG
   // the same network as SCL:
   IF "PLC2_Manual_Mode_Active" AND NOT "V3242_Xa_Bon3_Man" THEN "V3242_Xa_Bon3" := FALSE; END_IF;
END_REGION

REGION Network 36: Manual V3243_Xa_Bon3 - Set
   RUNG wire#powerrail
      Contact( "PLC2_Manual_Mode_Active" )
      Contact( "V3243_Xa_Bon3_Man" )
      S_Coil( "V3243_Xa_Bon3" )
   END_RUNG
   // the same network as SCL:
   IF "PLC2_Manual_Mode_Active" AND "V3243_Xa_Bon3_Man" THEN "V3243_Xa_Bon3" := TRUE; END_IF;
END_REGION

REGION Network 37: Manual V3243_Xa_Bon3 - Reset
   RUNG wire#powerrail
      Contact( "PLC2_Manual_Mode_Active" )
      I_Contact( "V3243_Xa_Bon3_Man" )
      R_Coil( "V3243_Xa_Bon3" )
   END_RUNG
   // the same network as SCL:
   IF "PLC2_Manual_Mode_Active" AND NOT "V3243_Xa_Bon3_Man" THEN "V3243_Xa_Bon3" := FALSE; END_IF;
END_REGION

REGION Network 38: Manual V3244_Xa_Bon3 - Set
   RUNG wire#powerrail
      Contact( "PLC2_Manual_Mode_Active" )
      Contact( "V3244_Xa_Bon3_Man" )
      S_Coil( "V3244_Xa_Bon3" )
   END_RUNG
   // the same network as SCL:
   IF "PLC2_Manual_Mode_Active" AND "V3244_Xa_Bon3_Man" THEN "V3244_Xa_Bon3" := TRUE; END_IF;
END_REGION

REGION Network 39: Manual V3244_Xa_Bon3 - Reset
   RUNG wire#powerrail
      Contact( "PLC2_Manual_Mode_Active" )
      I_Contact( "V3244_Xa_Bon3_Man" )
      R_Coil( "V3244_Xa_Bon3" )
   END_RUNG
   // the same network as SCL:
   IF "PLC2_Manual_Mode_Active" AND NOT "V3244_Xa_Bon3_Man" THEN "V3244_Xa_Bon3" := FALSE; END_IF;
END_REGION

REGION Network 40: Manual V3245_Nuoc_Bon4 - Set
   RUNG wire#powerrail
      Contact( "PLC2_Manual_Mode_Active" )
      Contact( "V3245_Nuoc_Bon4_Man" )
      S_Coil( "V3245_Nuoc_Bon4" )
   END_RUNG
   // the same network as SCL:
   IF "PLC2_Manual_Mode_Active" AND "V3245_Nuoc_Bon4_Man" THEN "V3245_Nuoc_Bon4" := TRUE; END_IF;
END_REGION

REGION Network 41: Manual V3245_Nuoc_Bon4 - Reset
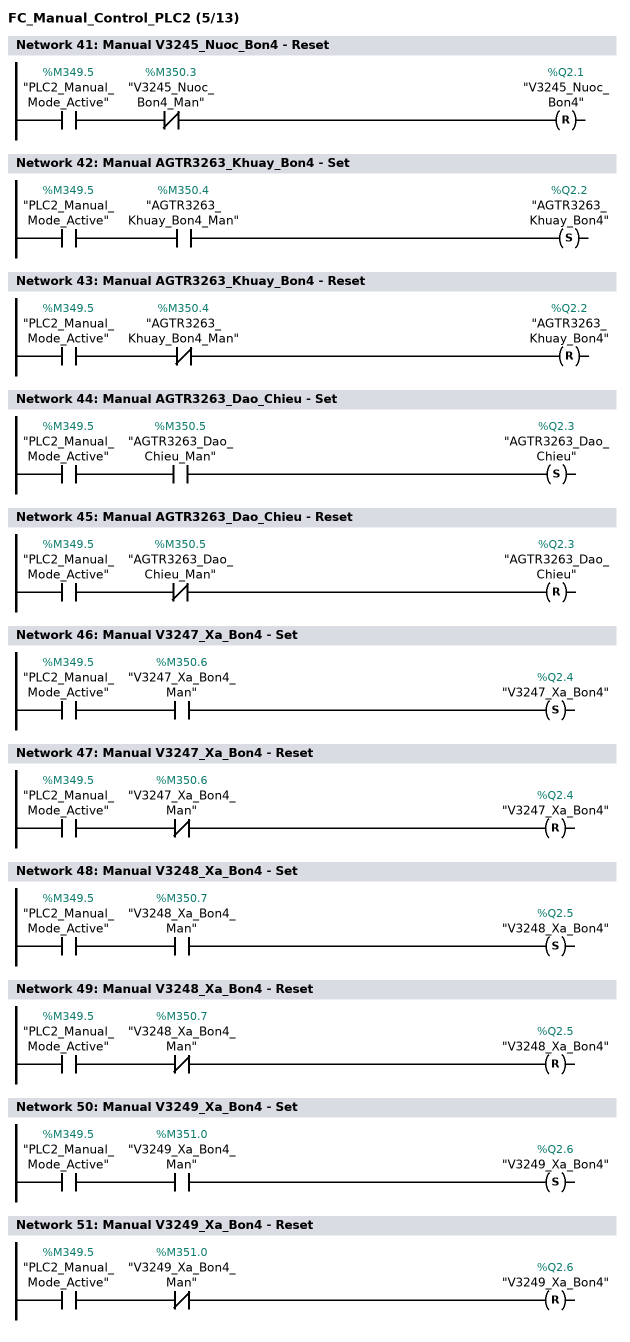
   RUNG wire#powerrail
      Contact( "PLC2_Manual_Mode_Active" )
      I_Contact( "V3245_Nuoc_Bon4_Man" )
      R_Coil( "V3245_Nuoc_Bon4" )
   END_RUNG
   // the same network as SCL:
   IF "PLC2_Manual_Mode_Active" AND NOT "V3245_Nuoc_Bon4_Man" THEN "V3245_Nuoc_Bon4" := FALSE; END_IF;
END_REGION

REGION Network 42: Manual AGTR3263_Khuay_Bon4 - Set
   RUNG wire#powerrail
      Contact( "PLC2_Manual_Mode_Active" )
      Contact( "AGTR3263_Khuay_Bon4_Man" )
      S_Coil( "AGTR3263_Khuay_Bon4" )
   END_RUNG
   // the same network as SCL:
   IF "PLC2_Manual_Mode_Active" AND "AGTR3263_Khuay_Bon4_Man" THEN "AGTR3263_Khuay_Bon4" := TRUE; END_IF;
END_REGION

REGION Network 43: Manual AGTR3263_Khuay_Bon4 - Reset
   RUNG wire#powerrail
      Contact( "PLC2_Manual_Mode_Active" )
      I_Contact( "AGTR3263_Khuay_Bon4_Man" )
      R_Coil( "AGTR3263_Khuay_Bon4" )
   END_RUNG
   // the same network as SCL:
   IF "PLC2_Manual_Mode_Active" AND NOT "AGTR3263_Khuay_Bon4_Man" THEN
       "AGTR3263_Khuay_Bon4" := FALSE;
   END_IF;
END_REGION

REGION Network 44: Manual AGTR3263_Dao_Chieu - Set
   RUNG wire#powerrail
      Contact( "PLC2_Manual_Mode_Active" )
      Contact( "AGTR3263_Dao_Chieu_Man" )
      S_Coil( "AGTR3263_Dao_Chieu" )
   END_RUNG
   // the same network as SCL:
   IF "PLC2_Manual_Mode_Active" AND "AGTR3263_Dao_Chieu_Man" THEN "AGTR3263_Dao_Chieu" := TRUE; END_IF;
END_REGION

REGION Network 45: Manual AGTR3263_Dao_Chieu - Reset
   RUNG wire#powerrail
      Contact( "PLC2_Manual_Mode_Active" )
      I_Contact( "AGTR3263_Dao_Chieu_Man" )
      R_Coil( "AGTR3263_Dao_Chieu" )
   END_RUNG
   // the same network as SCL:
   IF "PLC2_Manual_Mode_Active" AND NOT "AGTR3263_Dao_Chieu_Man" THEN "AGTR3263_Dao_Chieu" := FALSE; END_IF;
END_REGION

REGION Network 46: Manual V3247_Xa_Bon4 - Set
   RUNG wire#powerrail
      Contact( "PLC2_Manual_Mode_Active" )
      Contact( "V3247_Xa_Bon4_Man" )
      S_Coil( "V3247_Xa_Bon4" )
   END_RUNG
   // the same network as SCL:
   IF "PLC2_Manual_Mode_Active" AND "V3247_Xa_Bon4_Man" THEN "V3247_Xa_Bon4" := TRUE; END_IF;
END_REGION

REGION Network 47: Manual V3247_Xa_Bon4 - Reset
   RUNG wire#powerrail
      Contact( "PLC2_Manual_Mode_Active" )
      I_Contact( "V3247_Xa_Bon4_Man" )
      R_Coil( "V3247_Xa_Bon4" )
   END_RUNG
   // the same network as SCL:
   IF "PLC2_Manual_Mode_Active" AND NOT "V3247_Xa_Bon4_Man" THEN "V3247_Xa_Bon4" := FALSE; END_IF;
END_REGION

REGION Network 48: Manual V3248_Xa_Bon4 - Set
   RUNG wire#powerrail
      Contact( "PLC2_Manual_Mode_Active" )
      Contact( "V3248_Xa_Bon4_Man" )
      S_Coil( "V3248_Xa_Bon4" )
   END_RUNG
   // the same network as SCL:
   IF "PLC2_Manual_Mode_Active" AND "V3248_Xa_Bon4_Man" THEN "V3248_Xa_Bon4" := TRUE; END_IF;
END_REGION

REGION Network 49: Manual V3248_Xa_Bon4 - Reset
   RUNG wire#powerrail
      Contact( "PLC2_Manual_Mode_Active" )
      I_Contact( "V3248_Xa_Bon4_Man" )
      R_Coil( "V3248_Xa_Bon4" )
   END_RUNG
   // the same network as SCL:
   IF "PLC2_Manual_Mode_Active" AND NOT "V3248_Xa_Bon4_Man" THEN "V3248_Xa_Bon4" := FALSE; END_IF;
END_REGION

REGION Network 50: Manual V3249_Xa_Bon4 - Set
   RUNG wire#powerrail
      Contact( "PLC2_Manual_Mode_Active" )
      Contact( "V3249_Xa_Bon4_Man" )
      S_Coil( "V3249_Xa_Bon4" )
   END_RUNG
   // the same network as SCL:
   IF "PLC2_Manual_Mode_Active" AND "V3249_Xa_Bon4_Man" THEN "V3249_Xa_Bon4" := TRUE; END_IF;
END_REGION

REGION Network 51: Manual V3249_Xa_Bon4 - Reset
   RUNG wire#powerrail
      Contact( "PLC2_Manual_Mode_Active" )
      I_Contact( "V3249_Xa_Bon4_Man" )
      R_Coil( "V3249_Xa_Bon4" )
   END_RUNG
   // the same network as SCL:
   IF "PLC2_Manual_Mode_Active" AND NOT "V3249_Xa_Bon4_Man" THEN "V3249_Xa_Bon4" := FALSE; END_IF;
END_REGION

REGION Network 52: Manual CV3211_Nuoc_Bon3
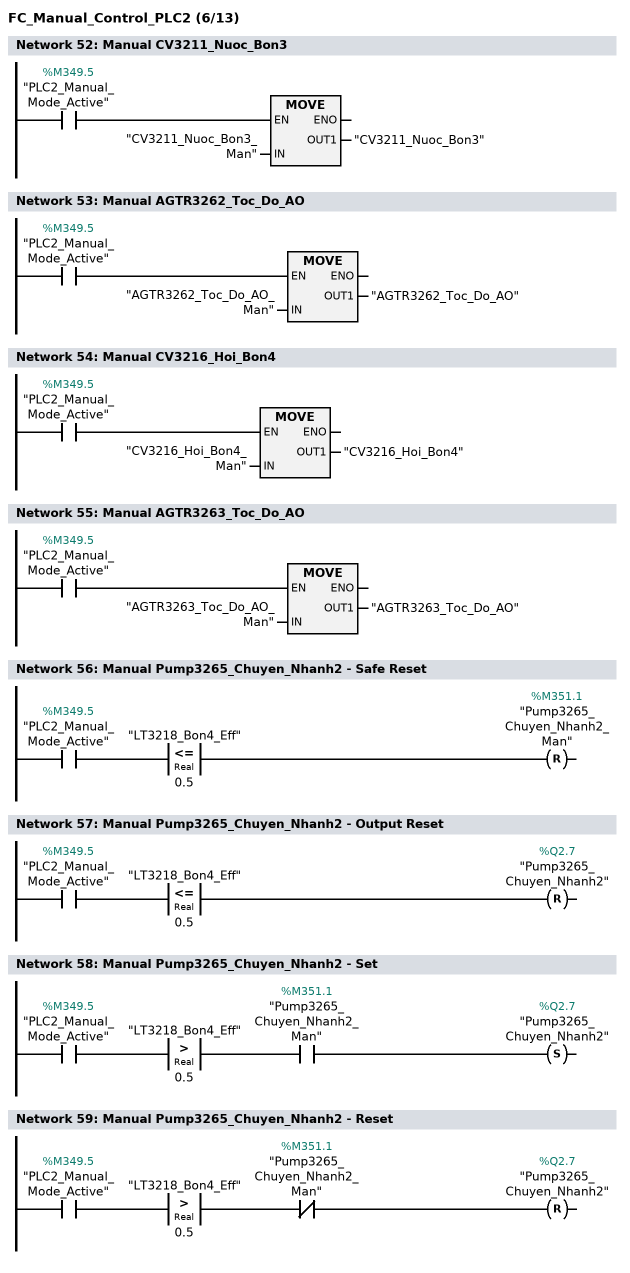
   RUNG wire#powerrail
      Contact( "PLC2_Manual_Mode_Active" )
      { S7_GenerateENO := "TRUE" } Move(in := "CV3211_Nuoc_Bon3_Man", out1 => "CV3211_Nuoc_Bon3")
   END_RUNG
   // the same network as SCL:
   IF "PLC2_Manual_Mode_Active" THEN "CV3211_Nuoc_Bon3" := "CV3211_Nuoc_Bon3_Man"; END_IF;
END_REGION

REGION Network 53: Manual AGTR3262_Toc_Do_AO
   RUNG wire#powerrail
      Contact( "PLC2_Manual_Mode_Active" )
      { S7_GenerateENO := "TRUE" } Move(in := "AGTR3262_Toc_Do_AO_Man", out1 => "AGTR3262_Toc_Do_AO")
   END_RUNG
   // the same network as SCL:
   IF "PLC2_Manual_Mode_Active" THEN "AGTR3262_Toc_Do_AO" := "AGTR3262_Toc_Do_AO_Man"; END_IF;
END_REGION

REGION Network 54: Manual CV3216_Hoi_Bon4
   RUNG wire#powerrail
      Contact( "PLC2_Manual_Mode_Active" )
      { S7_GenerateENO := "TRUE" } Move(in := "CV3216_Hoi_Bon4_Man", out1 => "CV3216_Hoi_Bon4")
   END_RUNG
   // the same network as SCL:
   IF "PLC2_Manual_Mode_Active" THEN "CV3216_Hoi_Bon4" := "CV3216_Hoi_Bon4_Man"; END_IF;
END_REGION

REGION Network 55: Manual AGTR3263_Toc_Do_AO
   RUNG wire#powerrail
      Contact( "PLC2_Manual_Mode_Active" )
      { S7_GenerateENO := "TRUE" } Move(in := "AGTR3263_Toc_Do_AO_Man", out1 => "AGTR3263_Toc_Do_AO")
   END_RUNG
   // the same network as SCL:
   IF "PLC2_Manual_Mode_Active" THEN "AGTR3263_Toc_Do_AO" := "AGTR3263_Toc_Do_AO_Man"; END_IF;
END_REGION

REGION Network 56: Manual Pump3265_Chuyen_Nhanh2 - Safe Reset
   RUNG wire#powerrail
      Contact( "PLC2_Manual_Mode_Active" )
      { S7_Templates := "SrcType := Real" } LE_Contact(in1 := "LT3218_Bon4_Eff", in2 := 0.5)
      R_Coil( "Pump3265_Chuyen_Nhanh2_Man" )
   END_RUNG
   // the same network as SCL:
   IF "PLC2_Manual_Mode_Active" AND ("LT3218_Bon4_Eff" <= 0.5) THEN
       "Pump3265_Chuyen_Nhanh2_Man" := FALSE;
   END_IF;
END_REGION

REGION Network 57: Manual Pump3265_Chuyen_Nhanh2 - Output Reset
   RUNG wire#powerrail
      Contact( "PLC2_Manual_Mode_Active" )
      { S7_Templates := "SrcType := Real" } LE_Contact(in1 := "LT3218_Bon4_Eff", in2 := 0.5)
      R_Coil( "Pump3265_Chuyen_Nhanh2" )
   END_RUNG
   // the same network as SCL:
   IF "PLC2_Manual_Mode_Active" AND ("LT3218_Bon4_Eff" <= 0.5) THEN
       "Pump3265_Chuyen_Nhanh2" := FALSE;
   END_IF;
END_REGION

REGION Network 58: Manual Pump3265_Chuyen_Nhanh2 - Set
   RUNG wire#powerrail
      Contact( "PLC2_Manual_Mode_Active" )
      { S7_Templates := "SrcType := Real" } GT_Contact(in1 := "LT3218_Bon4_Eff", in2 := 0.5)
      Contact( "Pump3265_Chuyen_Nhanh2_Man" )
      S_Coil( "Pump3265_Chuyen_Nhanh2" )
   END_RUNG
   // the same network as SCL:
   IF "PLC2_Manual_Mode_Active" AND ("LT3218_Bon4_Eff" > 0.5) AND "Pump3265_Chuyen_Nhanh2_Man" THEN
       "Pump3265_Chuyen_Nhanh2" := TRUE;
   END_IF;
END_REGION

REGION Network 59: Manual Pump3265_Chuyen_Nhanh2 - Reset
   RUNG wire#powerrail
      Contact( "PLC2_Manual_Mode_Active" )
      { S7_Templates := "SrcType := Real" } GT_Contact(in1 := "LT3218_Bon4_Eff", in2 := 0.5)
      I_Contact( "Pump3265_Chuyen_Nhanh2_Man" )
      R_Coil( "Pump3265_Chuyen_Nhanh2" )
   END_RUNG
   // the same network as SCL:
   IF "PLC2_Manual_Mode_Active" AND ("LT3218_Bon4_Eff" > 0.5) AND NOT "Pump3265_Chuyen_Nhanh2_Man" THEN
       "Pump3265_Chuyen_Nhanh2" := FALSE;
   END_IF;
END_REGION

REGION Network 60: Safety override - Reset V3240_Nuoc_Bon3
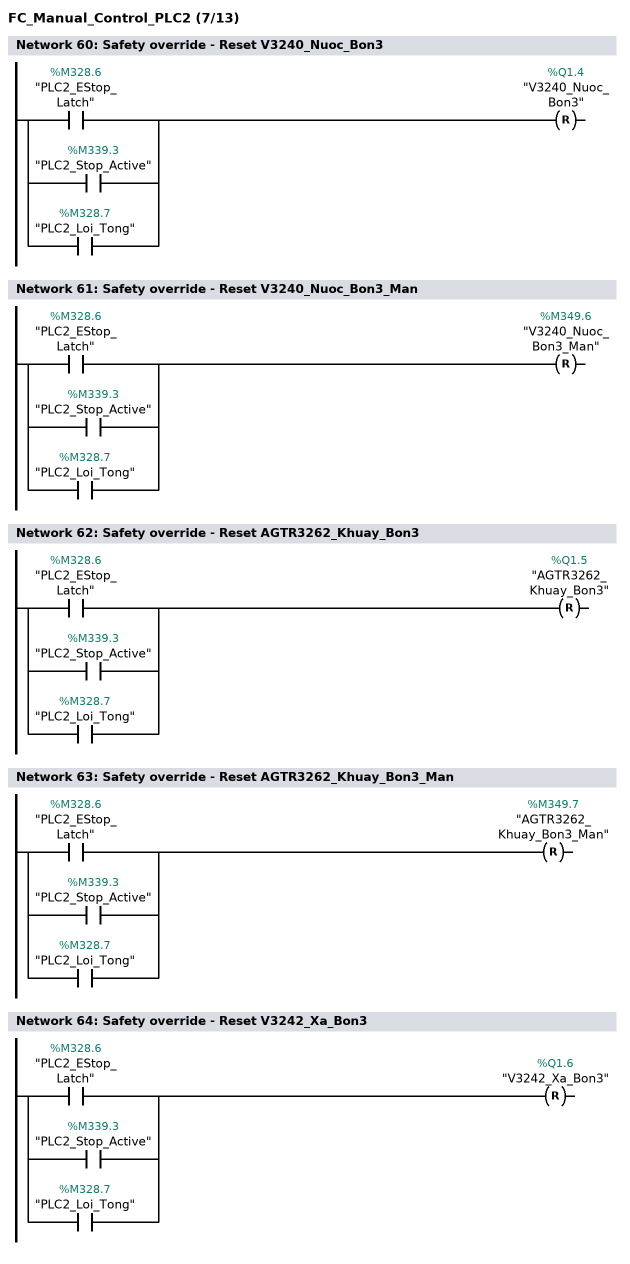
   RUNG wire#powerrail
      Contact( "PLC2_EStop_Latch" )
      wire#w1
      R_Coil( "V3240_Nuoc_Bon3" )
   END_RUNG
   RUNG wire#powerrail
      Contact( "PLC2_Stop_Active" )
   END_RUNG wire#w1
   RUNG wire#powerrail
      Contact( "PLC2_Loi_Tong" )
   END_RUNG wire#w1
   // the same network as SCL:
   IF "PLC2_EStop_Latch" OR "PLC2_Stop_Active" OR "PLC2_Loi_Tong" THEN "V3240_Nuoc_Bon3" := FALSE; END_IF;
END_REGION

REGION Network 61: Safety override - Reset V3240_Nuoc_Bon3_Man
   RUNG wire#powerrail
      Contact( "PLC2_EStop_Latch" )
      wire#w1
      R_Coil( "V3240_Nuoc_Bon3_Man" )
   END_RUNG
   RUNG wire#powerrail
      Contact( "PLC2_Stop_Active" )
   END_RUNG wire#w1
   RUNG wire#powerrail
      Contact( "PLC2_Loi_Tong" )
   END_RUNG wire#w1
   // the same network as SCL:
   IF "PLC2_EStop_Latch" OR "PLC2_Stop_Active" OR "PLC2_Loi_Tong" THEN
       "V3240_Nuoc_Bon3_Man" := FALSE;
   END_IF;
END_REGION

REGION Network 62: Safety override - Reset AGTR3262_Khuay_Bon3
   RUNG wire#powerrail
      Contact( "PLC2_EStop_Latch" )
      wire#w1
      R_Coil( "AGTR3262_Khuay_Bon3" )
   END_RUNG
   RUNG wire#powerrail
      Contact( "PLC2_Stop_Active" )
   END_RUNG wire#w1
   RUNG wire#powerrail
      Contact( "PLC2_Loi_Tong" )
   END_RUNG wire#w1
   // the same network as SCL:
   IF "PLC2_EStop_Latch" OR "PLC2_Stop_Active" OR "PLC2_Loi_Tong" THEN
       "AGTR3262_Khuay_Bon3" := FALSE;
   END_IF;
END_REGION

REGION Network 63: Safety override - Reset AGTR3262_Khuay_Bon3_Man
   RUNG wire#powerrail
      Contact( "PLC2_EStop_Latch" )
      wire#w1
      R_Coil( "AGTR3262_Khuay_Bon3_Man" )
   END_RUNG
   RUNG wire#powerrail
      Contact( "PLC2_Stop_Active" )
   END_RUNG wire#w1
   RUNG wire#powerrail
      Contact( "PLC2_Loi_Tong" )
   END_RUNG wire#w1
   // the same network as SCL:
   IF "PLC2_EStop_Latch" OR "PLC2_Stop_Active" OR "PLC2_Loi_Tong" THEN
       "AGTR3262_Khuay_Bon3_Man" := FALSE;
   END_IF;
END_REGION

REGION Network 64: Safety override - Reset V3242_Xa_Bon3
   RUNG wire#powerrail
      Contact( "PLC2_EStop_Latch" )
      wire#w1
      R_Coil( "V3242_Xa_Bon3" )
   END_RUNG
   RUNG wire#powerrail
      Contact( "PLC2_Stop_Active" )
   END_RUNG wire#w1
   RUNG wire#powerrail
      Contact( "PLC2_Loi_Tong" )
   END_RUNG wire#w1
   // the same network as SCL:
   IF "PLC2_EStop_Latch" OR "PLC2_Stop_Active" OR "PLC2_Loi_Tong" THEN "V3242_Xa_Bon3" := FALSE; END_IF;
END_REGION

REGION Network 65: Safety override - Reset V3242_Xa_Bon3_Man
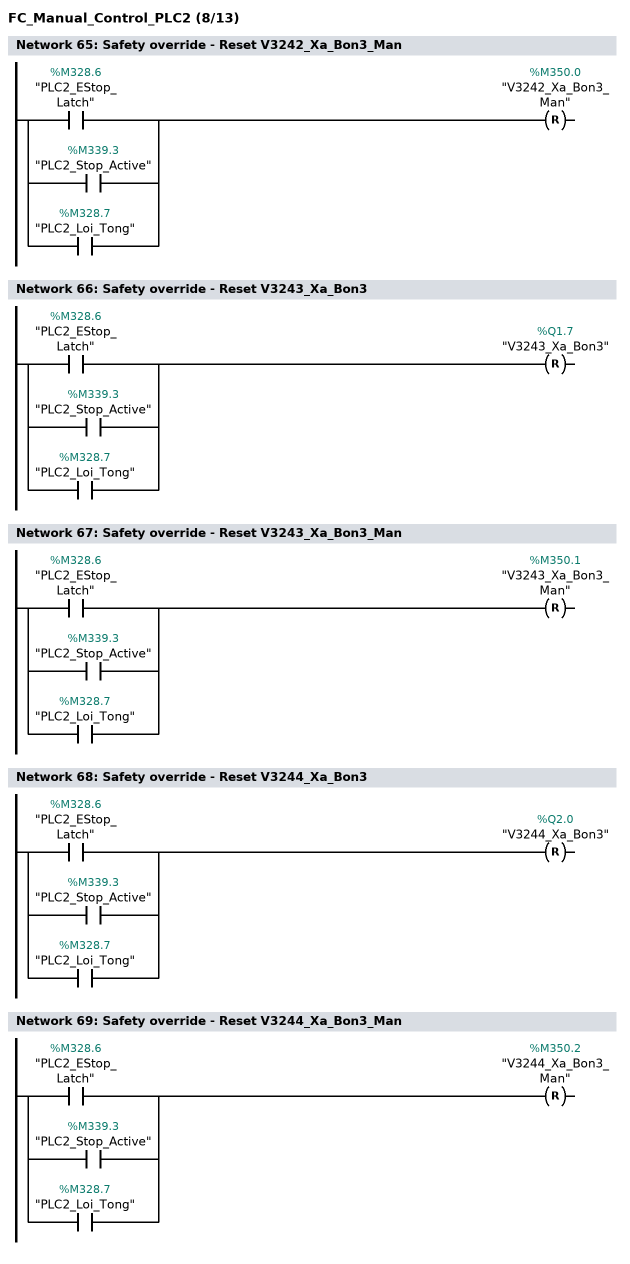
   RUNG wire#powerrail
      Contact( "PLC2_EStop_Latch" )
      wire#w1
      R_Coil( "V3242_Xa_Bon3_Man" )
   END_RUNG
   RUNG wire#powerrail
      Contact( "PLC2_Stop_Active" )
   END_RUNG wire#w1
   RUNG wire#powerrail
      Contact( "PLC2_Loi_Tong" )
   END_RUNG wire#w1
   // the same network as SCL:
   IF "PLC2_EStop_Latch" OR "PLC2_Stop_Active" OR "PLC2_Loi_Tong" THEN "V3242_Xa_Bon3_Man" := FALSE; END_IF;
END_REGION

REGION Network 66: Safety override - Reset V3243_Xa_Bon3
   RUNG wire#powerrail
      Contact( "PLC2_EStop_Latch" )
      wire#w1
      R_Coil( "V3243_Xa_Bon3" )
   END_RUNG
   RUNG wire#powerrail
      Contact( "PLC2_Stop_Active" )
   END_RUNG wire#w1
   RUNG wire#powerrail
      Contact( "PLC2_Loi_Tong" )
   END_RUNG wire#w1
   // the same network as SCL:
   IF "PLC2_EStop_Latch" OR "PLC2_Stop_Active" OR "PLC2_Loi_Tong" THEN "V3243_Xa_Bon3" := FALSE; END_IF;
END_REGION

REGION Network 67: Safety override - Reset V3243_Xa_Bon3_Man
   RUNG wire#powerrail
      Contact( "PLC2_EStop_Latch" )
      wire#w1
      R_Coil( "V3243_Xa_Bon3_Man" )
   END_RUNG
   RUNG wire#powerrail
      Contact( "PLC2_Stop_Active" )
   END_RUNG wire#w1
   RUNG wire#powerrail
      Contact( "PLC2_Loi_Tong" )
   END_RUNG wire#w1
   // the same network as SCL:
   IF "PLC2_EStop_Latch" OR "PLC2_Stop_Active" OR "PLC2_Loi_Tong" THEN "V3243_Xa_Bon3_Man" := FALSE; END_IF;
END_REGION

REGION Network 68: Safety override - Reset V3244_Xa_Bon3
   RUNG wire#powerrail
      Contact( "PLC2_EStop_Latch" )
      wire#w1
      R_Coil( "V3244_Xa_Bon3" )
   END_RUNG
   RUNG wire#powerrail
      Contact( "PLC2_Stop_Active" )
   END_RUNG wire#w1
   RUNG wire#powerrail
      Contact( "PLC2_Loi_Tong" )
   END_RUNG wire#w1
   // the same network as SCL:
   IF "PLC2_EStop_Latch" OR "PLC2_Stop_Active" OR "PLC2_Loi_Tong" THEN "V3244_Xa_Bon3" := FALSE; END_IF;
END_REGION

REGION Network 69: Safety override - Reset V3244_Xa_Bon3_Man
   RUNG wire#powerrail
      Contact( "PLC2_EStop_Latch" )
      wire#w1
      R_Coil( "V3244_Xa_Bon3_Man" )
   END_RUNG
   RUNG wire#powerrail
      Contact( "PLC2_Stop_Active" )
   END_RUNG wire#w1
   RUNG wire#powerrail
      Contact( "PLC2_Loi_Tong" )
   END_RUNG wire#w1
   // the same network as SCL:
   IF "PLC2_EStop_Latch" OR "PLC2_Stop_Active" OR "PLC2_Loi_Tong" THEN "V3244_Xa_Bon3_Man" := FALSE; END_IF;
END_REGION

REGION Network 70: Safety override - Reset V3245_Nuoc_Bon4
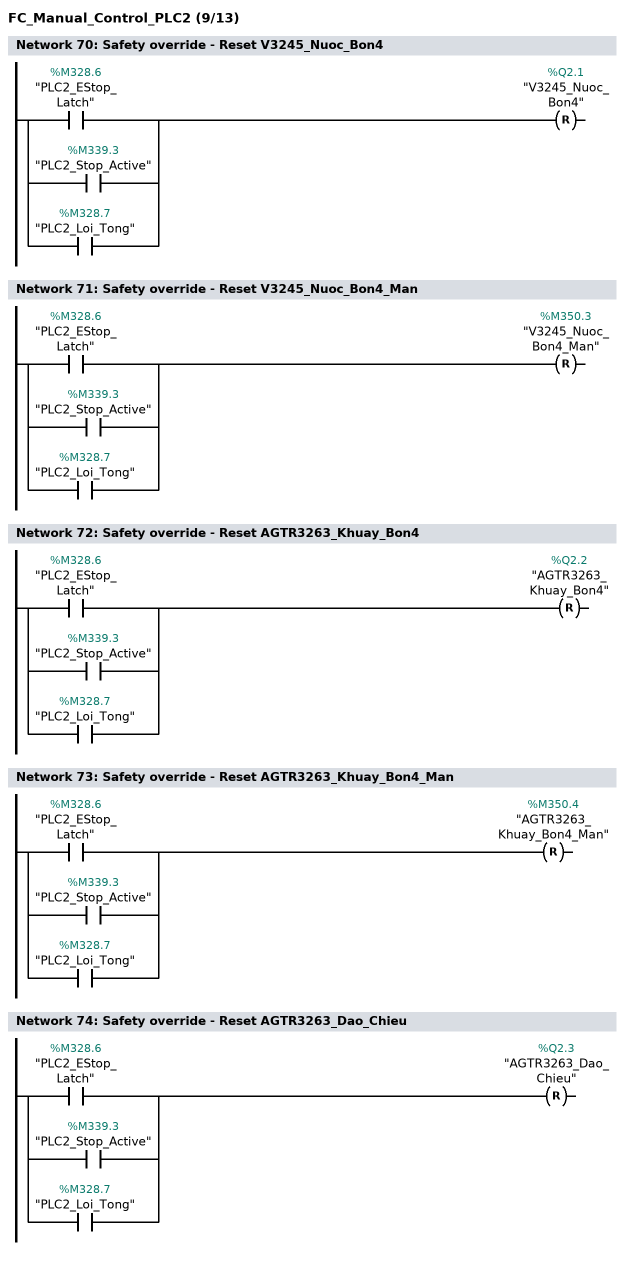
   RUNG wire#powerrail
      Contact( "PLC2_EStop_Latch" )
      wire#w1
      R_Coil( "V3245_Nuoc_Bon4" )
   END_RUNG
   RUNG wire#powerrail
      Contact( "PLC2_Stop_Active" )
   END_RUNG wire#w1
   RUNG wire#powerrail
      Contact( "PLC2_Loi_Tong" )
   END_RUNG wire#w1
   // the same network as SCL:
   IF "PLC2_EStop_Latch" OR "PLC2_Stop_Active" OR "PLC2_Loi_Tong" THEN "V3245_Nuoc_Bon4" := FALSE; END_IF;
END_REGION

REGION Network 71: Safety override - Reset V3245_Nuoc_Bon4_Man
   RUNG wire#powerrail
      Contact( "PLC2_EStop_Latch" )
      wire#w1
      R_Coil( "V3245_Nuoc_Bon4_Man" )
   END_RUNG
   RUNG wire#powerrail
      Contact( "PLC2_Stop_Active" )
   END_RUNG wire#w1
   RUNG wire#powerrail
      Contact( "PLC2_Loi_Tong" )
   END_RUNG wire#w1
   // the same network as SCL:
   IF "PLC2_EStop_Latch" OR "PLC2_Stop_Active" OR "PLC2_Loi_Tong" THEN
       "V3245_Nuoc_Bon4_Man" := FALSE;
   END_IF;
END_REGION

REGION Network 72: Safety override - Reset AGTR3263_Khuay_Bon4
   RUNG wire#powerrail
      Contact( "PLC2_EStop_Latch" )
      wire#w1
      R_Coil( "AGTR3263_Khuay_Bon4" )
   END_RUNG
   RUNG wire#powerrail
      Contact( "PLC2_Stop_Active" )
   END_RUNG wire#w1
   RUNG wire#powerrail
      Contact( "PLC2_Loi_Tong" )
   END_RUNG wire#w1
   // the same network as SCL:
   IF "PLC2_EStop_Latch" OR "PLC2_Stop_Active" OR "PLC2_Loi_Tong" THEN
       "AGTR3263_Khuay_Bon4" := FALSE;
   END_IF;
END_REGION

REGION Network 73: Safety override - Reset AGTR3263_Khuay_Bon4_Man
   RUNG wire#powerrail
      Contact( "PLC2_EStop_Latch" )
      wire#w1
      R_Coil( "AGTR3263_Khuay_Bon4_Man" )
   END_RUNG
   RUNG wire#powerrail
      Contact( "PLC2_Stop_Active" )
   END_RUNG wire#w1
   RUNG wire#powerrail
      Contact( "PLC2_Loi_Tong" )
   END_RUNG wire#w1
   // the same network as SCL:
   IF "PLC2_EStop_Latch" OR "PLC2_Stop_Active" OR "PLC2_Loi_Tong" THEN
       "AGTR3263_Khuay_Bon4_Man" := FALSE;
   END_IF;
END_REGION

REGION Network 74: Safety override - Reset AGTR3263_Dao_Chieu
   RUNG wire#powerrail
      Contact( "PLC2_EStop_Latch" )
      wire#w1
      R_Coil( "AGTR3263_Dao_Chieu" )
   END_RUNG
   RUNG wire#powerrail
      Contact( "PLC2_Stop_Active" )
   END_RUNG wire#w1
   RUNG wire#powerrail
      Contact( "PLC2_Loi_Tong" )
   END_RUNG wire#w1
   // the same network as SCL:
   IF "PLC2_EStop_Latch" OR "PLC2_Stop_Active" OR "PLC2_Loi_Tong" THEN "AGTR3263_Dao_Chieu" := FALSE; END_IF;
END_REGION

REGION Network 75: Safety override - Reset AGTR3263_Dao_Chieu_Man
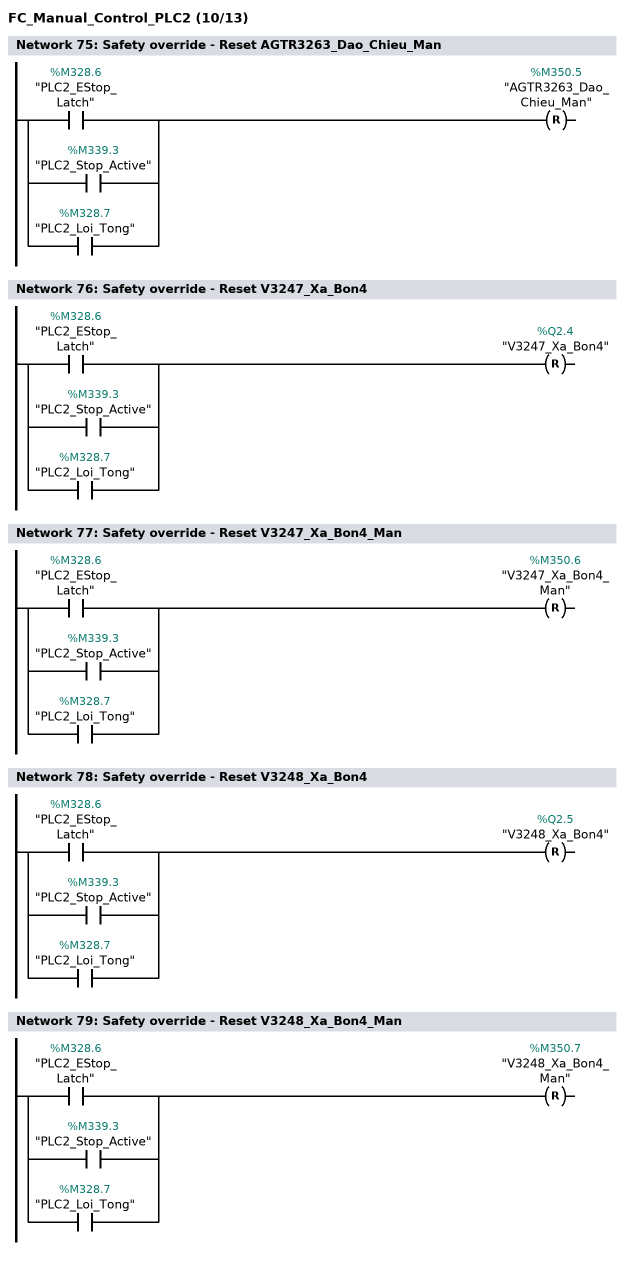
   RUNG wire#powerrail
      Contact( "PLC2_EStop_Latch" )
      wire#w1
      R_Coil( "AGTR3263_Dao_Chieu_Man" )
   END_RUNG
   RUNG wire#powerrail
      Contact( "PLC2_Stop_Active" )
   END_RUNG wire#w1
   RUNG wire#powerrail
      Contact( "PLC2_Loi_Tong" )
   END_RUNG wire#w1
   // the same network as SCL:
   IF "PLC2_EStop_Latch" OR "PLC2_Stop_Active" OR "PLC2_Loi_Tong" THEN
       "AGTR3263_Dao_Chieu_Man" := FALSE;
   END_IF;
END_REGION

REGION Network 76: Safety override - Reset V3247_Xa_Bon4
   RUNG wire#powerrail
      Contact( "PLC2_EStop_Latch" )
      wire#w1
      R_Coil( "V3247_Xa_Bon4" )
   END_RUNG
   RUNG wire#powerrail
      Contact( "PLC2_Stop_Active" )
   END_RUNG wire#w1
   RUNG wire#powerrail
      Contact( "PLC2_Loi_Tong" )
   END_RUNG wire#w1
   // the same network as SCL:
   IF "PLC2_EStop_Latch" OR "PLC2_Stop_Active" OR "PLC2_Loi_Tong" THEN "V3247_Xa_Bon4" := FALSE; END_IF;
END_REGION

REGION Network 77: Safety override - Reset V3247_Xa_Bon4_Man
   RUNG wire#powerrail
      Contact( "PLC2_EStop_Latch" )
      wire#w1
      R_Coil( "V3247_Xa_Bon4_Man" )
   END_RUNG
   RUNG wire#powerrail
      Contact( "PLC2_Stop_Active" )
   END_RUNG wire#w1
   RUNG wire#powerrail
      Contact( "PLC2_Loi_Tong" )
   END_RUNG wire#w1
   // the same network as SCL:
   IF "PLC2_EStop_Latch" OR "PLC2_Stop_Active" OR "PLC2_Loi_Tong" THEN "V3247_Xa_Bon4_Man" := FALSE; END_IF;
END_REGION

REGION Network 78: Safety override - Reset V3248_Xa_Bon4
   RUNG wire#powerrail
      Contact( "PLC2_EStop_Latch" )
      wire#w1
      R_Coil( "V3248_Xa_Bon4" )
   END_RUNG
   RUNG wire#powerrail
      Contact( "PLC2_Stop_Active" )
   END_RUNG wire#w1
   RUNG wire#powerrail
      Contact( "PLC2_Loi_Tong" )
   END_RUNG wire#w1
   // the same network as SCL:
   IF "PLC2_EStop_Latch" OR "PLC2_Stop_Active" OR "PLC2_Loi_Tong" THEN "V3248_Xa_Bon4" := FALSE; END_IF;
END_REGION

REGION Network 79: Safety override - Reset V3248_Xa_Bon4_Man
   RUNG wire#powerrail
      Contact( "PLC2_EStop_Latch" )
      wire#w1
      R_Coil( "V3248_Xa_Bon4_Man" )
   END_RUNG
   RUNG wire#powerrail
      Contact( "PLC2_Stop_Active" )
   END_RUNG wire#w1
   RUNG wire#powerrail
      Contact( "PLC2_Loi_Tong" )
   END_RUNG wire#w1
   // the same network as SCL:
   IF "PLC2_EStop_Latch" OR "PLC2_Stop_Active" OR "PLC2_Loi_Tong" THEN "V3248_Xa_Bon4_Man" := FALSE; END_IF;
END_REGION

REGION Network 80: Safety override - Reset V3249_Xa_Bon4
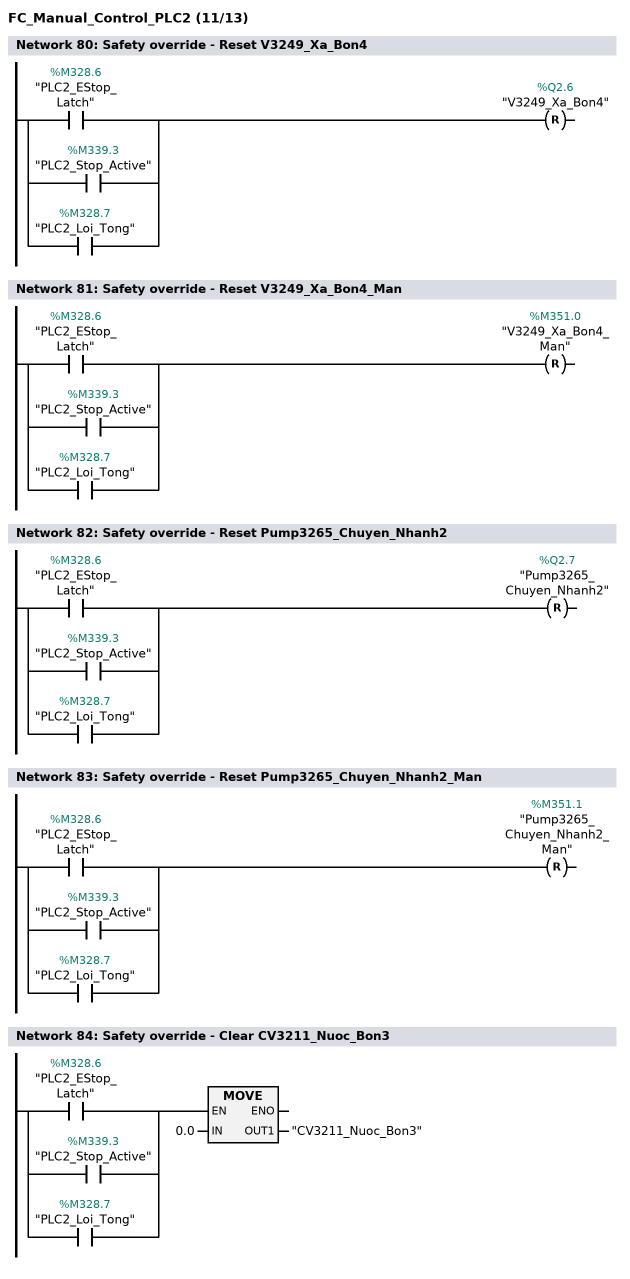
   RUNG wire#powerrail
      Contact( "PLC2_EStop_Latch" )
      wire#w1
      R_Coil( "V3249_Xa_Bon4" )
   END_RUNG
   RUNG wire#powerrail
      Contact( "PLC2_Stop_Active" )
   END_RUNG wire#w1
   RUNG wire#powerrail
      Contact( "PLC2_Loi_Tong" )
   END_RUNG wire#w1
   // the same network as SCL:
   IF "PLC2_EStop_Latch" OR "PLC2_Stop_Active" OR "PLC2_Loi_Tong" THEN "V3249_Xa_Bon4" := FALSE; END_IF;
END_REGION

REGION Network 81: Safety override - Reset V3249_Xa_Bon4_Man
   RUNG wire#powerrail
      Contact( "PLC2_EStop_Latch" )
      wire#w1
      R_Coil( "V3249_Xa_Bon4_Man" )
   END_RUNG
   RUNG wire#powerrail
      Contact( "PLC2_Stop_Active" )
   END_RUNG wire#w1
   RUNG wire#powerrail
      Contact( "PLC2_Loi_Tong" )
   END_RUNG wire#w1
   // the same network as SCL:
   IF "PLC2_EStop_Latch" OR "PLC2_Stop_Active" OR "PLC2_Loi_Tong" THEN "V3249_Xa_Bon4_Man" := FALSE; END_IF;
END_REGION

REGION Network 82: Safety override - Reset Pump3265_Chuyen_Nhanh2
   RUNG wire#powerrail
      Contact( "PLC2_EStop_Latch" )
      wire#w1
      R_Coil( "Pump3265_Chuyen_Nhanh2" )
   END_RUNG
   RUNG wire#powerrail
      Contact( "PLC2_Stop_Active" )
   END_RUNG wire#w1
   RUNG wire#powerrail
      Contact( "PLC2_Loi_Tong" )
   END_RUNG wire#w1
   // the same network as SCL:
   IF "PLC2_EStop_Latch" OR "PLC2_Stop_Active" OR "PLC2_Loi_Tong" THEN
       "Pump3265_Chuyen_Nhanh2" := FALSE;
   END_IF;
END_REGION

REGION Network 83: Safety override - Reset Pump3265_Chuyen_Nhanh2_Man
   RUNG wire#powerrail
      Contact( "PLC2_EStop_Latch" )
      wire#w1
      R_Coil( "Pump3265_Chuyen_Nhanh2_Man" )
   END_RUNG
   RUNG wire#powerrail
      Contact( "PLC2_Stop_Active" )
   END_RUNG wire#w1
   RUNG wire#powerrail
      Contact( "PLC2_Loi_Tong" )
   END_RUNG wire#w1
   // the same network as SCL:
   IF "PLC2_EStop_Latch" OR "PLC2_Stop_Active" OR "PLC2_Loi_Tong" THEN
       "Pump3265_Chuyen_Nhanh2_Man" := FALSE;
   END_IF;
END_REGION

REGION Network 84: Safety override - Clear CV3211_Nuoc_Bon3
   RUNG wire#powerrail
      Contact( "PLC2_EStop_Latch" )
      wire#w1
      { S7_GenerateENO := "TRUE" } Move(in := 0.0, out1 => "CV3211_Nuoc_Bon3")
   END_RUNG
   RUNG wire#powerrail
      Contact( "PLC2_Stop_Active" )
   END_RUNG wire#w1
   RUNG wire#powerrail
      Contact( "PLC2_Loi_Tong" )
   END_RUNG wire#w1
   // the same network as SCL:
   IF "PLC2_EStop_Latch" OR "PLC2_Stop_Active" OR "PLC2_Loi_Tong" THEN "CV3211_Nuoc_Bon3" := 0.0; END_IF;
END_REGION

REGION Network 85: Safety override - Clear CV3211_Nuoc_Bon3_Man
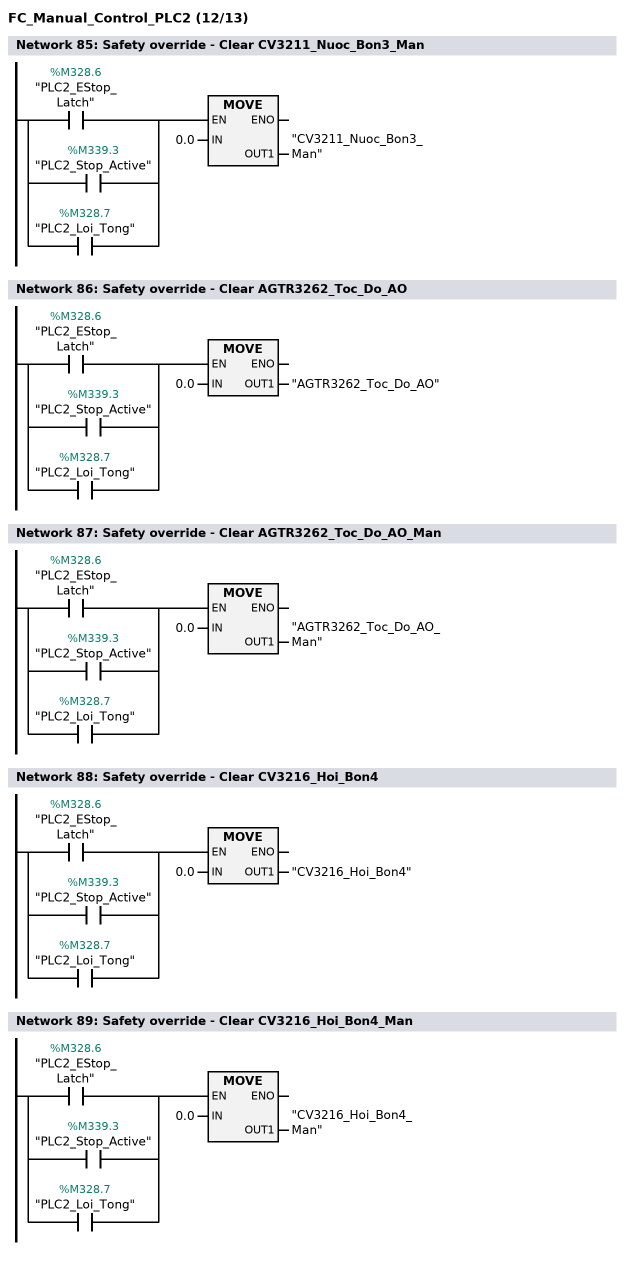
   RUNG wire#powerrail
      Contact( "PLC2_EStop_Latch" )
      wire#w1
      { S7_GenerateENO := "TRUE" } Move(in := 0.0, out1 => "CV3211_Nuoc_Bon3_Man")
   END_RUNG
   RUNG wire#powerrail
      Contact( "PLC2_Stop_Active" )
   END_RUNG wire#w1
   RUNG wire#powerrail
      Contact( "PLC2_Loi_Tong" )
   END_RUNG wire#w1
   // the same network as SCL:
   IF "PLC2_EStop_Latch" OR "PLC2_Stop_Active" OR "PLC2_Loi_Tong" THEN "CV3211_Nuoc_Bon3_Man" := 0.0; END_IF;
END_REGION

REGION Network 86: Safety override - Clear AGTR3262_Toc_Do_AO
   RUNG wire#powerrail
      Contact( "PLC2_EStop_Latch" )
      wire#w1
      { S7_GenerateENO := "TRUE" } Move(in := 0.0, out1 => "AGTR3262_Toc_Do_AO")
   END_RUNG
   RUNG wire#powerrail
      Contact( "PLC2_Stop_Active" )
   END_RUNG wire#w1
   RUNG wire#powerrail
      Contact( "PLC2_Loi_Tong" )
   END_RUNG wire#w1
   // the same network as SCL:
   IF "PLC2_EStop_Latch" OR "PLC2_Stop_Active" OR "PLC2_Loi_Tong" THEN "AGTR3262_Toc_Do_AO" := 0.0; END_IF;
END_REGION

REGION Network 87: Safety override - Clear AGTR3262_Toc_Do_AO_Man
   RUNG wire#powerrail
      Contact( "PLC2_EStop_Latch" )
      wire#w1
      { S7_GenerateENO := "TRUE" } Move(in := 0.0, out1 => "AGTR3262_Toc_Do_AO_Man")
   END_RUNG
   RUNG wire#powerrail
      Contact( "PLC2_Stop_Active" )
   END_RUNG wire#w1
   RUNG wire#powerrail
      Contact( "PLC2_Loi_Tong" )
   END_RUNG wire#w1
   // the same network as SCL:
   IF "PLC2_EStop_Latch" OR "PLC2_Stop_Active" OR "PLC2_Loi_Tong" THEN
       "AGTR3262_Toc_Do_AO_Man" := 0.0;
   END_IF;
END_REGION

REGION Network 88: Safety override - Clear CV3216_Hoi_Bon4
   RUNG wire#powerrail
      Contact( "PLC2_EStop_Latch" )
      wire#w1
      { S7_GenerateENO := "TRUE" } Move(in := 0.0, out1 => "CV3216_Hoi_Bon4")
   END_RUNG
   RUNG wire#powerrail
      Contact( "PLC2_Stop_Active" )
   END_RUNG wire#w1
   RUNG wire#powerrail
      Contact( "PLC2_Loi_Tong" )
   END_RUNG wire#w1
   // the same network as SCL:
   IF "PLC2_EStop_Latch" OR "PLC2_Stop_Active" OR "PLC2_Loi_Tong" THEN "CV3216_Hoi_Bon4" := 0.0; END_IF;
END_REGION

REGION Network 89: Safety override - Clear CV3216_Hoi_Bon4_Man
   RUNG wire#powerrail
      Contact( "PLC2_EStop_Latch" )
      wire#w1
      { S7_GenerateENO := "TRUE" } Move(in := 0.0, out1 => "CV3216_Hoi_Bon4_Man")
   END_RUNG
   RUNG wire#powerrail
      Contact( "PLC2_Stop_Active" )
   END_RUNG wire#w1
   RUNG wire#powerrail
      Contact( "PLC2_Loi_Tong" )
   END_RUNG wire#w1
   // the same network as SCL:
   IF "PLC2_EStop_Latch" OR "PLC2_Stop_Active" OR "PLC2_Loi_Tong" THEN "CV3216_Hoi_Bon4_Man" := 0.0; END_IF;
END_REGION

REGION Network 90: Safety override - Clear AGTR3263_Toc_Do_AO
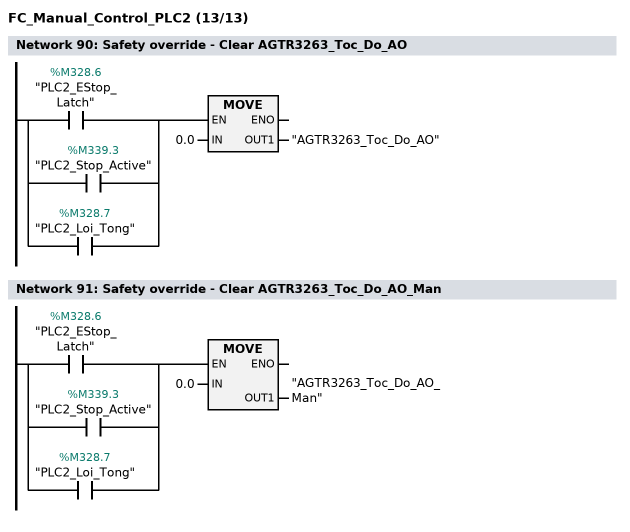
   RUNG wire#powerrail
      Contact( "PLC2_EStop_Latch" )
      wire#w1
      { S7_GenerateENO := "TRUE" } Move(in := 0.0, out1 => "AGTR3263_Toc_Do_AO")
   END_RUNG
   RUNG wire#powerrail
      Contact( "PLC2_Stop_Active" )
   END_RUNG wire#w1
   RUNG wire#powerrail
      Contact( "PLC2_Loi_Tong" )
   END_RUNG wire#w1
   // the same network as SCL:
   IF "PLC2_EStop_Latch" OR "PLC2_Stop_Active" OR "PLC2_Loi_Tong" THEN "AGTR3263_Toc_Do_AO" := 0.0; END_IF;
END_REGION

REGION Network 91: Safety override - Clear AGTR3263_Toc_Do_AO_Man
   RUNG wire#powerrail
      Contact( "PLC2_EStop_Latch" )
      wire#w1
      { S7_GenerateENO := "TRUE" } Move(in := 0.0, out1 => "AGTR3263_Toc_Do_AO_Man")
   END_RUNG
   RUNG wire#powerrail
      Contact( "PLC2_Stop_Active" )
   END_RUNG wire#w1
   RUNG wire#powerrail
      Contact( "PLC2_Loi_Tong" )
   END_RUNG wire#w1
   // the same network as SCL:
   IF "PLC2_EStop_Latch" OR "PLC2_Stop_Active" OR "PLC2_Loi_Tong" THEN
       "AGTR3263_Toc_Do_AO_Man" := 0.0;
   END_IF;
END_REGION
END_FUNCTION

FUNCTION "FC_HMI_Mirror_PLC2" : Void   // FC41, LAD
{ S7_Optimized_Access := 'TRUE' }
VERSION : 0.1
// stored: AutoNumber true, IsIECCheckEnabled false, SetENOAutomatically false, UDAEnableTagReadback false
BEGIN

REGION Network 1: Mirror V3240_Nuoc_Bon3
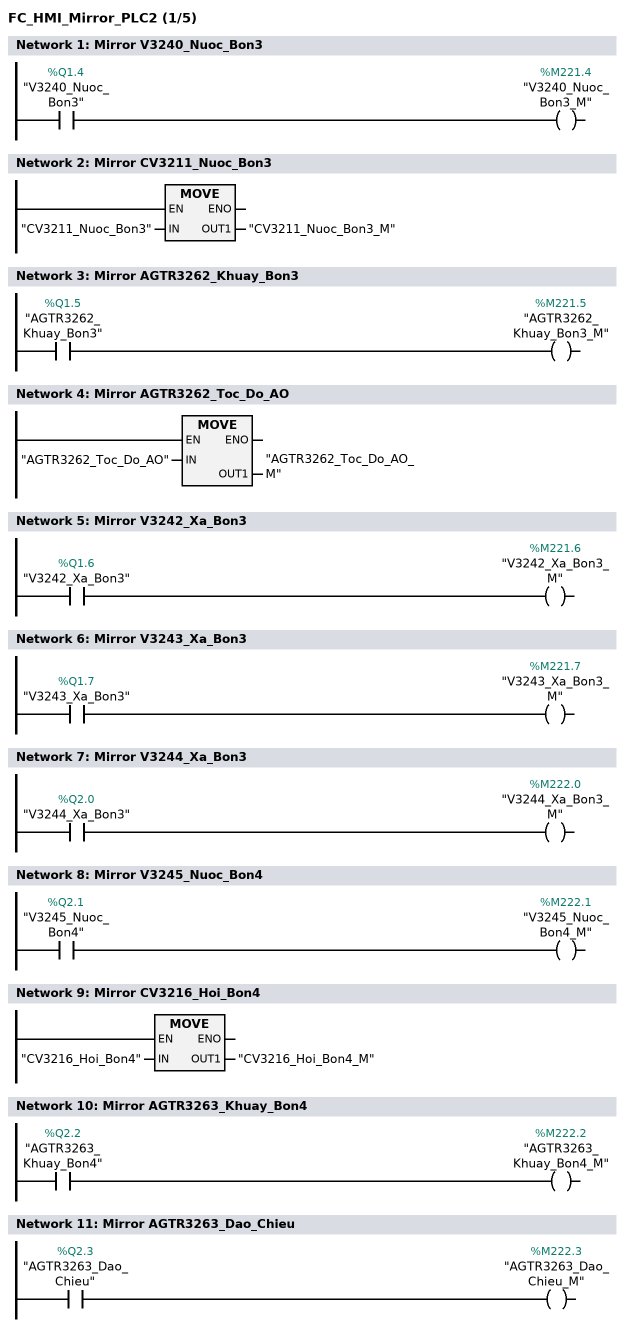
   RUNG wire#powerrail
      Contact( "V3240_Nuoc_Bon3" )
      Coil( "V3240_Nuoc_Bon3_M" )
   END_RUNG
   // the same network as SCL:
   "V3240_Nuoc_Bon3_M" := "V3240_Nuoc_Bon3";
END_REGION

REGION Network 2: Mirror CV3211_Nuoc_Bon3
   RUNG wire#powerrail
      { S7_GenerateENO := "TRUE" } Move(in := "CV3211_Nuoc_Bon3", out1 => "CV3211_Nuoc_Bon3_M")
   END_RUNG
   // the same network as SCL:
   "CV3211_Nuoc_Bon3_M" := "CV3211_Nuoc_Bon3";
END_REGION

REGION Network 3: Mirror AGTR3262_Khuay_Bon3
   RUNG wire#powerrail
      Contact( "AGTR3262_Khuay_Bon3" )
      Coil( "AGTR3262_Khuay_Bon3_M" )
   END_RUNG
   // the same network as SCL:
   "AGTR3262_Khuay_Bon3_M" := "AGTR3262_Khuay_Bon3";
END_REGION

REGION Network 4: Mirror AGTR3262_Toc_Do_AO
   RUNG wire#powerrail
      { S7_GenerateENO := "TRUE" } Move(in := "AGTR3262_Toc_Do_AO", out1 => "AGTR3262_Toc_Do_AO_M")
   END_RUNG
   // the same network as SCL:
   "AGTR3262_Toc_Do_AO_M" := "AGTR3262_Toc_Do_AO";
END_REGION

REGION Network 5: Mirror V3242_Xa_Bon3
   RUNG wire#powerrail
      Contact( "V3242_Xa_Bon3" )
      Coil( "V3242_Xa_Bon3_M" )
   END_RUNG
   // the same network as SCL:
   "V3242_Xa_Bon3_M" := "V3242_Xa_Bon3";
END_REGION

REGION Network 6: Mirror V3243_Xa_Bon3
   RUNG wire#powerrail
      Contact( "V3243_Xa_Bon3" )
      Coil( "V3243_Xa_Bon3_M" )
   END_RUNG
   // the same network as SCL:
   "V3243_Xa_Bon3_M" := "V3243_Xa_Bon3";
END_REGION

REGION Network 7: Mirror V3244_Xa_Bon3
   RUNG wire#powerrail
      Contact( "V3244_Xa_Bon3" )
      Coil( "V3244_Xa_Bon3_M" )
   END_RUNG
   // the same network as SCL:
   "V3244_Xa_Bon3_M" := "V3244_Xa_Bon3";
END_REGION

REGION Network 8: Mirror V3245_Nuoc_Bon4
   RUNG wire#powerrail
      Contact( "V3245_Nuoc_Bon4" )
      Coil( "V3245_Nuoc_Bon4_M" )
   END_RUNG
   // the same network as SCL:
   "V3245_Nuoc_Bon4_M" := "V3245_Nuoc_Bon4";
END_REGION

REGION Network 9: Mirror CV3216_Hoi_Bon4
   RUNG wire#powerrail
      { S7_GenerateENO := "TRUE" } Move(in := "CV3216_Hoi_Bon4", out1 => "CV3216_Hoi_Bon4_M")
   END_RUNG
   // the same network as SCL:
   "CV3216_Hoi_Bon4_M" := "CV3216_Hoi_Bon4";
END_REGION

REGION Network 10: Mirror AGTR3263_Khuay_Bon4
   RUNG wire#powerrail
      Contact( "AGTR3263_Khuay_Bon4" )
      Coil( "AGTR3263_Khuay_Bon4_M" )
   END_RUNG
   // the same network as SCL:
   "AGTR3263_Khuay_Bon4_M" := "AGTR3263_Khuay_Bon4";
END_REGION

REGION Network 11: Mirror AGTR3263_Dao_Chieu
   RUNG wire#powerrail
      Contact( "AGTR3263_Dao_Chieu" )
      Coil( "AGTR3263_Dao_Chieu_M" )
   END_RUNG
   // the same network as SCL:
   "AGTR3263_Dao_Chieu_M" := "AGTR3263_Dao_Chieu";
END_REGION

REGION Network 12: Mirror AGTR3263_Toc_Do_AO
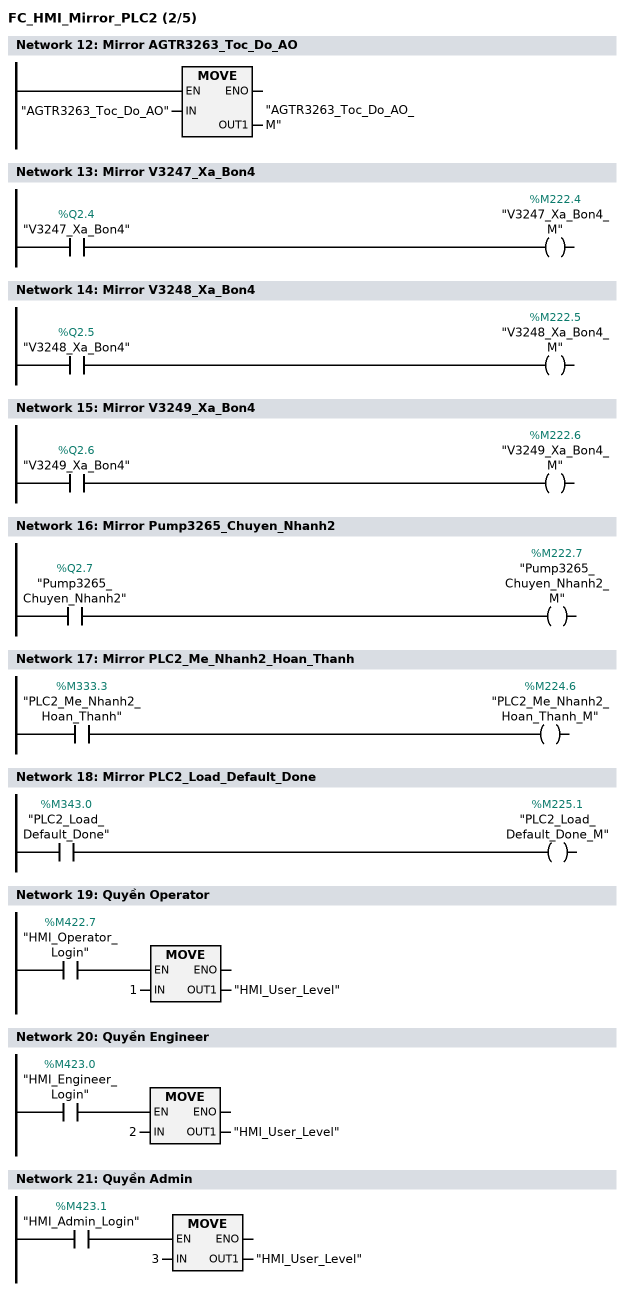
   RUNG wire#powerrail
      { S7_GenerateENO := "TRUE" } Move(in := "AGTR3263_Toc_Do_AO", out1 => "AGTR3263_Toc_Do_AO_M")
   END_RUNG
   // the same network as SCL:
   "AGTR3263_Toc_Do_AO_M" := "AGTR3263_Toc_Do_AO";
END_REGION

REGION Network 13: Mirror V3247_Xa_Bon4
   RUNG wire#powerrail
      Contact( "V3247_Xa_Bon4" )
      Coil( "V3247_Xa_Bon4_M" )
   END_RUNG
   // the same network as SCL:
   "V3247_Xa_Bon4_M" := "V3247_Xa_Bon4";
END_REGION

REGION Network 14: Mirror V3248_Xa_Bon4
   RUNG wire#powerrail
      Contact( "V3248_Xa_Bon4" )
      Coil( "V3248_Xa_Bon4_M" )
   END_RUNG
   // the same network as SCL:
   "V3248_Xa_Bon4_M" := "V3248_Xa_Bon4";
END_REGION

REGION Network 15: Mirror V3249_Xa_Bon4
   RUNG wire#powerrail
      Contact( "V3249_Xa_Bon4" )
      Coil( "V3249_Xa_Bon4_M" )
   END_RUNG
   // the same network as SCL:
   "V3249_Xa_Bon4_M" := "V3249_Xa_Bon4";
END_REGION

REGION Network 16: Mirror Pump3265_Chuyen_Nhanh2
   RUNG wire#powerrail
      Contact( "Pump3265_Chuyen_Nhanh2" )
      Coil( "Pump3265_Chuyen_Nhanh2_M" )
   END_RUNG
   // the same network as SCL:
   "Pump3265_Chuyen_Nhanh2_M" := "Pump3265_Chuyen_Nhanh2";
END_REGION

REGION Network 17: Mirror PLC2_Me_Nhanh2_Hoan_Thanh
   RUNG wire#powerrail
      Contact( "PLC2_Me_Nhanh2_Hoan_Thanh" )
      Coil( "PLC2_Me_Nhanh2_Hoan_Thanh_M" )
   END_RUNG
   // the same network as SCL:
   "PLC2_Me_Nhanh2_Hoan_Thanh_M" := "PLC2_Me_Nhanh2_Hoan_Thanh";
END_REGION

REGION Network 18: Mirror PLC2_Load_Default_Done
   RUNG wire#powerrail
      Contact( "PLC2_Load_Default_Done" )
      Coil( "PLC2_Load_Default_Done_M" )
   END_RUNG
   // the same network as SCL:
   "PLC2_Load_Default_Done_M" := "PLC2_Load_Default_Done";
END_REGION

REGION Network 19: Quyền Operator
   RUNG wire#powerrail
      Contact( "HMI_Operator_Login" )
      { S7_GenerateENO := "TRUE" } Move(in := 1, out1 => "HMI_User_Level")
   END_RUNG
   // the same network as SCL:
   IF "HMI_Operator_Login" THEN "HMI_User_Level" := 1; END_IF;
END_REGION

REGION Network 20: Quyền Engineer
   RUNG wire#powerrail
      Contact( "HMI_Engineer_Login" )
      { S7_GenerateENO := "TRUE" } Move(in := 2, out1 => "HMI_User_Level")
   END_RUNG
   // the same network as SCL:
   IF "HMI_Engineer_Login" THEN "HMI_User_Level" := 2; END_IF;
END_REGION

REGION Network 21: Quyền Admin
   RUNG wire#powerrail
      Contact( "HMI_Admin_Login" )
      { S7_GenerateENO := "TRUE" } Move(in := 3, out1 => "HMI_User_Level")
   END_RUNG
   // the same network as SCL:
   IF "HMI_Admin_Login" THEN "HMI_User_Level" := 3; END_IF;
END_REGION

REGION Network 22: Cho phép sửa thông số Engineer
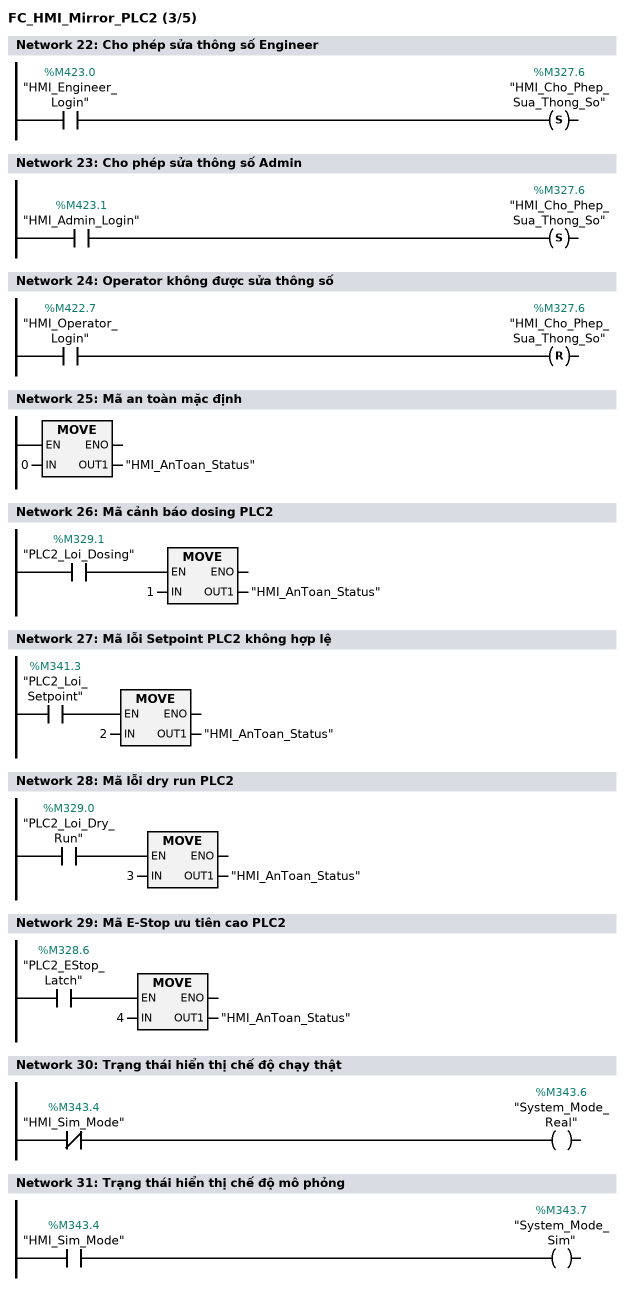
   RUNG wire#powerrail
      Contact( "HMI_Engineer_Login" )
      S_Coil( "HMI_Cho_Phep_Sua_Thong_So" )
   END_RUNG
   // the same network as SCL:
   IF "HMI_Engineer_Login" THEN "HMI_Cho_Phep_Sua_Thong_So" := TRUE; END_IF;
END_REGION

REGION Network 23: Cho phép sửa thông số Admin
   RUNG wire#powerrail
      Contact( "HMI_Admin_Login" )
      S_Coil( "HMI_Cho_Phep_Sua_Thong_So" )
   END_RUNG
   // the same network as SCL:
   IF "HMI_Admin_Login" THEN "HMI_Cho_Phep_Sua_Thong_So" := TRUE; END_IF;
END_REGION

REGION Network 24: Operator không được sửa thông số
   RUNG wire#powerrail
      Contact( "HMI_Operator_Login" )
      R_Coil( "HMI_Cho_Phep_Sua_Thong_So" )
   END_RUNG
   // the same network as SCL:
   IF "HMI_Operator_Login" THEN "HMI_Cho_Phep_Sua_Thong_So" := FALSE; END_IF;
END_REGION

REGION Network 25: Mã an toàn mặc định
   RUNG wire#powerrail
      { S7_GenerateENO := "TRUE" } Move(in := 0, out1 => "HMI_AnToan_Status")
   END_RUNG
   // the same network as SCL:
   "HMI_AnToan_Status" := 0;
END_REGION

REGION Network 26: Mã cảnh báo dosing PLC2
   RUNG wire#powerrail
      Contact( "PLC2_Loi_Dosing" )
      { S7_GenerateENO := "TRUE" } Move(in := 1, out1 => "HMI_AnToan_Status")
   END_RUNG
   // the same network as SCL:
   IF "PLC2_Loi_Dosing" THEN "HMI_AnToan_Status" := 1; END_IF;
END_REGION

REGION Network 27: Mã lỗi Setpoint PLC2 không hợp lệ
   RUNG wire#powerrail
      Contact( "PLC2_Loi_Setpoint" )
      { S7_GenerateENO := "TRUE" } Move(in := 2, out1 => "HMI_AnToan_Status")
   END_RUNG
   // the same network as SCL:
   IF "PLC2_Loi_Setpoint" THEN "HMI_AnToan_Status" := 2; END_IF;
END_REGION

REGION Network 28: Mã lỗi dry run PLC2
   RUNG wire#powerrail
      Contact( "PLC2_Loi_Dry_Run" )
      { S7_GenerateENO := "TRUE" } Move(in := 3, out1 => "HMI_AnToan_Status")
   END_RUNG
   // the same network as SCL:
   IF "PLC2_Loi_Dry_Run" THEN "HMI_AnToan_Status" := 3; END_IF;
END_REGION

REGION Network 29: Mã E-Stop ưu tiên cao PLC2
   RUNG wire#powerrail
      Contact( "PLC2_EStop_Latch" )
      { S7_GenerateENO := "TRUE" } Move(in := 4, out1 => "HMI_AnToan_Status")
   END_RUNG
   // the same network as SCL:
   IF "PLC2_EStop_Latch" THEN "HMI_AnToan_Status" := 4; END_IF;
END_REGION

REGION Network 30: Trạng thái hiển thị chế độ chạy thật
   RUNG wire#powerrail
      I_Contact( "HMI_Sim_Mode" )
      Coil( "System_Mode_Real" )
   END_RUNG
   // the same network as SCL:
   "System_Mode_Real" := NOT "HMI_Sim_Mode";
END_REGION

REGION Network 31: Trạng thái hiển thị chế độ mô phỏng
   RUNG wire#powerrail
      Contact( "HMI_Sim_Mode" )
      Coil( "System_Mode_Sim" )
   END_RUNG
   // the same network as SCL:
   "System_Mode_Sim" := "HMI_Sim_Mode";
END_REGION

REGION Network 32: Cảnh báo chế độ mô phỏng HMI active
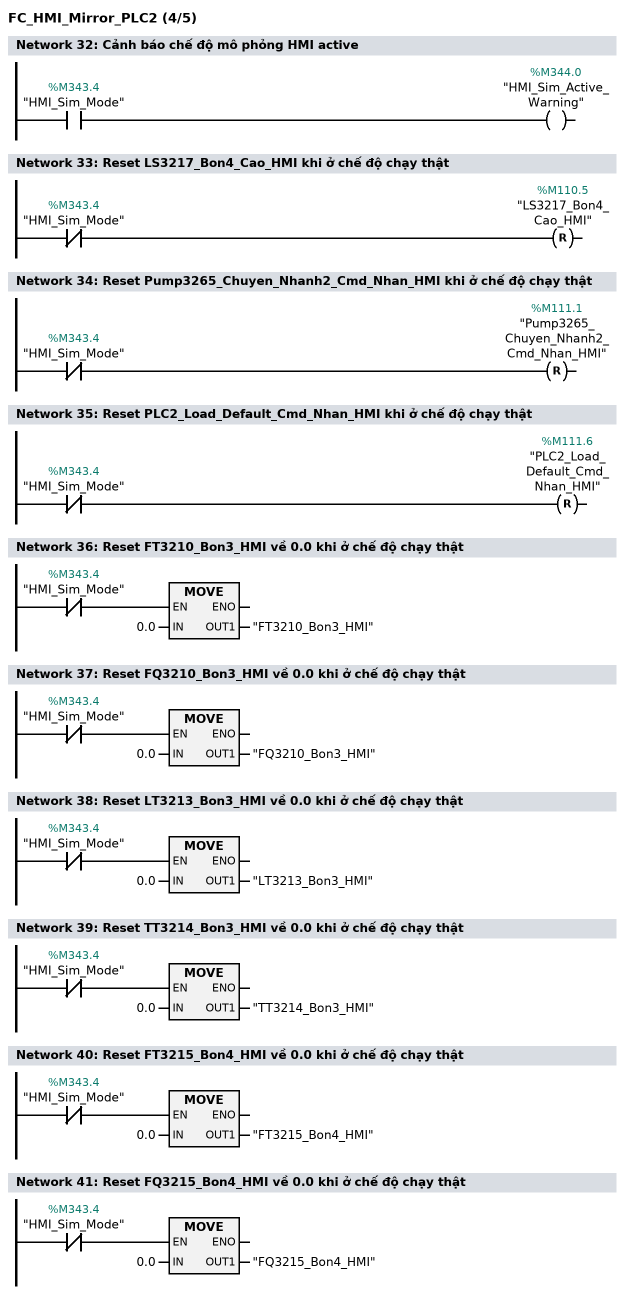
   RUNG wire#powerrail
      Contact( "HMI_Sim_Mode" )
      Coil( "HMI_Sim_Active_Warning" )
   END_RUNG
   // the same network as SCL:
   "HMI_Sim_Active_Warning" := "HMI_Sim_Mode";
END_REGION

REGION Network 33: Reset LS3217_Bon4_Cao_HMI khi ở chế độ chạy thật
   RUNG wire#powerrail
      I_Contact( "HMI_Sim_Mode" )
      R_Coil( "LS3217_Bon4_Cao_HMI" )
   END_RUNG
   // the same network as SCL:
   IF NOT "HMI_Sim_Mode" THEN "LS3217_Bon4_Cao_HMI" := FALSE; END_IF;
END_REGION

REGION Network 34: Reset Pump3265_Chuyen_Nhanh2_Cmd_Nhan_HMI khi ở chế độ chạy thật
   RUNG wire#powerrail
      I_Contact( "HMI_Sim_Mode" )
      R_Coil( "Pump3265_Chuyen_Nhanh2_Cmd_Nhan_HMI" )
   END_RUNG
   // the same network as SCL:
   IF NOT "HMI_Sim_Mode" THEN "Pump3265_Chuyen_Nhanh2_Cmd_Nhan_HMI" := FALSE; END_IF;
END_REGION

REGION Network 35: Reset PLC2_Load_Default_Cmd_Nhan_HMI khi ở chế độ chạy thật
   RUNG wire#powerrail
      I_Contact( "HMI_Sim_Mode" )
      R_Coil( "PLC2_Load_Default_Cmd_Nhan_HMI" )
   END_RUNG
   // the same network as SCL:
   IF NOT "HMI_Sim_Mode" THEN "PLC2_Load_Default_Cmd_Nhan_HMI" := FALSE; END_IF;
END_REGION

REGION Network 36: Reset FT3210_Bon3_HMI về 0.0 khi ở chế độ chạy thật
   RUNG wire#powerrail
      I_Contact( "HMI_Sim_Mode" )
      { S7_GenerateENO := "TRUE" } Move(in := 0.0, out1 => "FT3210_Bon3_HMI")
   END_RUNG
   // the same network as SCL:
   IF NOT "HMI_Sim_Mode" THEN "FT3210_Bon3_HMI" := 0.0; END_IF;
END_REGION

REGION Network 37: Reset FQ3210_Bon3_HMI về 0.0 khi ở chế độ chạy thật
   RUNG wire#powerrail
      I_Contact( "HMI_Sim_Mode" )
      { S7_GenerateENO := "TRUE" } Move(in := 0.0, out1 => "FQ3210_Bon3_HMI")
   END_RUNG
   // the same network as SCL:
   IF NOT "HMI_Sim_Mode" THEN "FQ3210_Bon3_HMI" := 0.0; END_IF;
END_REGION

REGION Network 38: Reset LT3213_Bon3_HMI về 0.0 khi ở chế độ chạy thật
   RUNG wire#powerrail
      I_Contact( "HMI_Sim_Mode" )
      { S7_GenerateENO := "TRUE" } Move(in := 0.0, out1 => "LT3213_Bon3_HMI")
   END_RUNG
   // the same network as SCL:
   IF NOT "HMI_Sim_Mode" THEN "LT3213_Bon3_HMI" := 0.0; END_IF;
END_REGION

REGION Network 39: Reset TT3214_Bon3_HMI về 0.0 khi ở chế độ chạy thật
   RUNG wire#powerrail
      I_Contact( "HMI_Sim_Mode" )
      { S7_GenerateENO := "TRUE" } Move(in := 0.0, out1 => "TT3214_Bon3_HMI")
   END_RUNG
   // the same network as SCL:
   IF NOT "HMI_Sim_Mode" THEN "TT3214_Bon3_HMI" := 0.0; END_IF;
END_REGION

REGION Network 40: Reset FT3215_Bon4_HMI về 0.0 khi ở chế độ chạy thật
   RUNG wire#powerrail
      I_Contact( "HMI_Sim_Mode" )
      { S7_GenerateENO := "TRUE" } Move(in := 0.0, out1 => "FT3215_Bon4_HMI")
   END_RUNG
   // the same network as SCL:
   IF NOT "HMI_Sim_Mode" THEN "FT3215_Bon4_HMI" := 0.0; END_IF;
END_REGION

REGION Network 41: Reset FQ3215_Bon4_HMI về 0.0 khi ở chế độ chạy thật
   RUNG wire#powerrail
      I_Contact( "HMI_Sim_Mode" )
      { S7_GenerateENO := "TRUE" } Move(in := 0.0, out1 => "FQ3215_Bon4_HMI")
   END_RUNG
   // the same network as SCL:
   IF NOT "HMI_Sim_Mode" THEN "FQ3215_Bon4_HMI" := 0.0; END_IF;
END_REGION

REGION Network 42: Reset LT3218_Bon4_HMI về 0.0 khi ở chế độ chạy thật
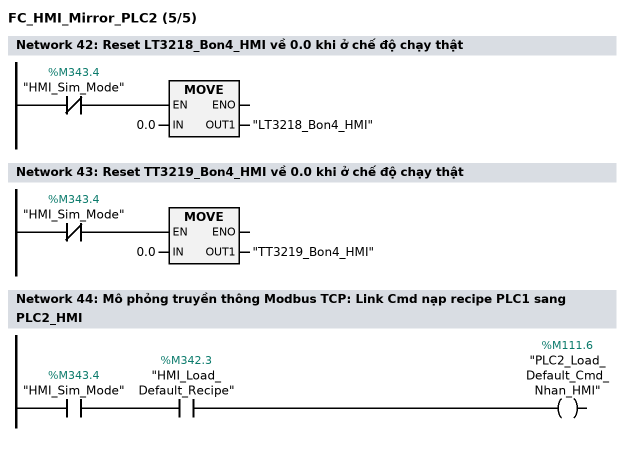
   RUNG wire#powerrail
      I_Contact( "HMI_Sim_Mode" )
      { S7_GenerateENO := "TRUE" } Move(in := 0.0, out1 => "LT3218_Bon4_HMI")
   END_RUNG
   // the same network as SCL:
   IF NOT "HMI_Sim_Mode" THEN "LT3218_Bon4_HMI" := 0.0; END_IF;
END_REGION

REGION Network 43: Reset TT3219_Bon4_HMI về 0.0 khi ở chế độ chạy thật
   RUNG wire#powerrail
      I_Contact( "HMI_Sim_Mode" )
      { S7_GenerateENO := "TRUE" } Move(in := 0.0, out1 => "TT3219_Bon4_HMI")
   END_RUNG
   // the same network as SCL:
   IF NOT "HMI_Sim_Mode" THEN "TT3219_Bon4_HMI" := 0.0; END_IF;
END_REGION

REGION Network 44: Mô phỏng truyền thông Modbus TCP: Link Cmd nạp recipe PLC1 sang PLC2_HMI
   RUNG wire#powerrail
      Contact( "HMI_Sim_Mode" )
      Contact( "HMI_Load_Default_Recipe" )
      Coil( "PLC2_Load_Default_Cmd_Nhan_HMI" )
   END_RUNG
   // the same network as SCL:
   "PLC2_Load_Default_Cmd_Nhan_HMI" := "HMI_Sim_Mode" AND "HMI_Load_Default_Recipe";
END_REGION
END_FUNCTION

ORGANIZATION_BLOCK "OB31_PID_PLC2_Bon4"   // OB31, LAD, CyclicInterrupt
{ S7_Optimized_Access := 'TRUE' }
VERSION : 0.1
// stored: AutoNumber true, IsIECCheckEnabled false, SetENOAutomatically false
   VAR_INPUT
      Initial_Call : Bool;   // Initial call of this OB
      Event_Count : Int;   // Events discarded
   END_VAR
BEGIN

REGION Network 1: Initialize PID Bon 4 Kp parameter
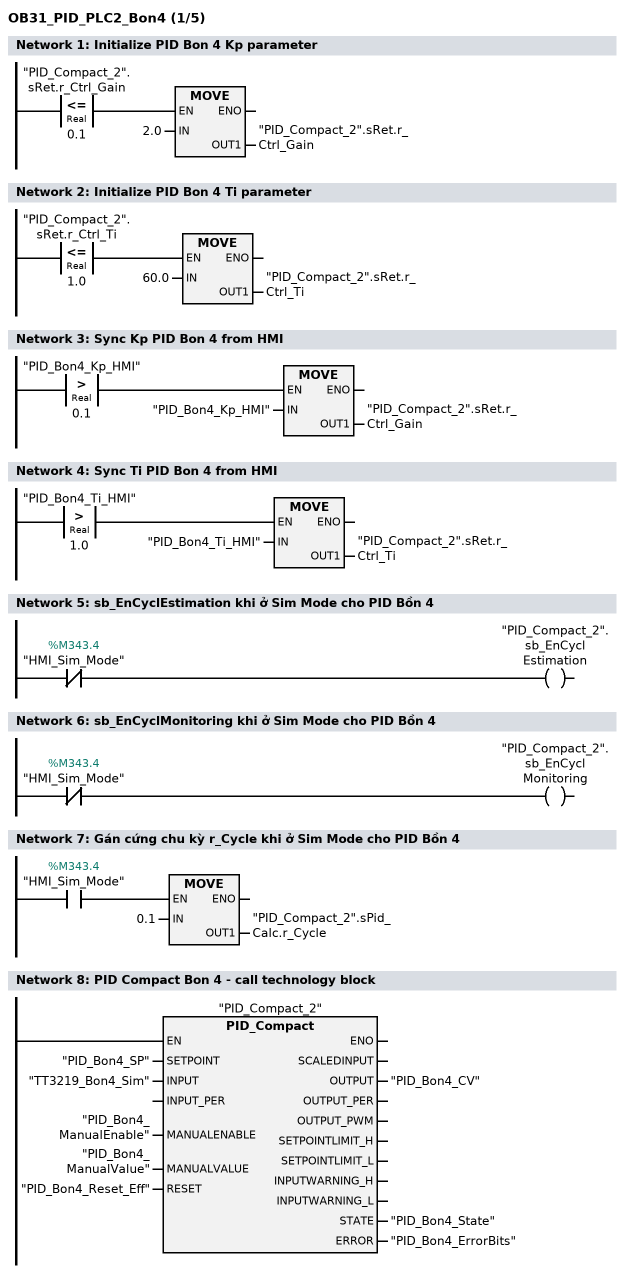
   RUNG wire#powerrail
      { S7_Templates := "SrcType := Real" } LE_Contact(in1 := "PID_Compact_2".sRet.r_Ctrl_Gain, in2 := 0.1)
      { S7_GenerateENO := "TRUE" } Move(in := 2.0, out1 => "PID_Compact_2".sRet.r_Ctrl_Gain)
   END_RUNG
   // the same network as SCL:
   IF "PID_Compact_2".sRet.r_Ctrl_Gain <= 0.1 THEN "PID_Compact_2".sRet.r_Ctrl_Gain := 2.0; END_IF;
END_REGION

REGION Network 2: Initialize PID Bon 4 Ti parameter
   RUNG wire#powerrail
      { S7_Templates := "SrcType := Real" } LE_Contact(in1 := "PID_Compact_2".sRet.r_Ctrl_Ti, in2 := 1.0)
      { S7_GenerateENO := "TRUE" } Move(in := 60.0, out1 => "PID_Compact_2".sRet.r_Ctrl_Ti)
   END_RUNG
   // the same network as SCL:
   IF "PID_Compact_2".sRet.r_Ctrl_Ti <= 1.0 THEN "PID_Compact_2".sRet.r_Ctrl_Ti := 60.0; END_IF;
END_REGION

REGION Network 3: Sync Kp PID Bon 4 from HMI
   RUNG wire#powerrail
      { S7_Templates := "SrcType := Real" } GT_Contact(in1 := "PID_Bon4_Kp_HMI", in2 := 0.1)
      { S7_GenerateENO := "TRUE" } Move(in := "PID_Bon4_Kp_HMI", out1 => "PID_Compact_2".sRet.r_Ctrl_Gain)
   END_RUNG
   // the same network as SCL:
   IF "PID_Bon4_Kp_HMI" > 0.1 THEN "PID_Compact_2".sRet.r_Ctrl_Gain := "PID_Bon4_Kp_HMI"; END_IF;
END_REGION

REGION Network 4: Sync Ti PID Bon 4 from HMI
   RUNG wire#powerrail
      { S7_Templates := "SrcType := Real" } GT_Contact(in1 := "PID_Bon4_Ti_HMI", in2 := 1.0)
      { S7_GenerateENO := "TRUE" } Move(in := "PID_Bon4_Ti_HMI", out1 => "PID_Compact_2".sRet.r_Ctrl_Ti)
   END_RUNG
   // the same network as SCL:
   IF "PID_Bon4_Ti_HMI" > 1.0 THEN "PID_Compact_2".sRet.r_Ctrl_Ti := "PID_Bon4_Ti_HMI"; END_IF;
END_REGION

REGION Network 5: sb_EnCyclEstimation khi ở Sim Mode cho PID Bồn 4
   RUNG wire#powerrail
      I_Contact( "HMI_Sim_Mode" )
      Coil( "PID_Compact_2".sb_EnCyclEstimation )
   END_RUNG
   // the same network as SCL:
   "PID_Compact_2".sb_EnCyclEstimation := NOT "HMI_Sim_Mode";
END_REGION

REGION Network 6: sb_EnCyclMonitoring khi ở Sim Mode cho PID Bồn 4
   RUNG wire#powerrail
      I_Contact( "HMI_Sim_Mode" )
      Coil( "PID_Compact_2".sb_EnCyclMonitoring )
   END_RUNG
   // the same network as SCL:
   "PID_Compact_2".sb_EnCyclMonitoring := NOT "HMI_Sim_Mode";
END_REGION

REGION Network 7: Gán cứng chu kỳ r_Cycle khi ở Sim Mode cho PID Bồn 4
   RUNG wire#powerrail
      Contact( "HMI_Sim_Mode" )
      { S7_GenerateENO := "TRUE" } Move(in := 0.1, out1 => "PID_Compact_2".sPid_Calc.r_Cycle)
   END_RUNG
   // the same network as SCL:
   IF "HMI_Sim_Mode" THEN "PID_Compact_2".sPid_Calc.r_Cycle := 0.1; END_IF;
END_REGION

REGION Network 8: PID Compact Bon 4 - call technology block
   RUNG wire#powerrail
      "PID_Compact_2".PID_Compact(Setpoint := "PID_Bon4_SP", Input := "TT3219_Bon4_Sim", Input_PER :=, ManualEnable := "PID_Bon4_ManualEnable", ManualValue := "PID_Bon4_ManualValue", Reset := "PID_Bon4_Reset_Eff", ScaledInput =>, Output => "PID_Bon4_CV", Output_PER =>, Output_PWM =>, SetpointLimit_H =>, SetpointLimit_L =>, InputWarning_H =>, InputWarning_L =>, State => "PID_Bon4_State", Error => "PID_Bon4_ErrorBits")
   END_RUNG
   // the same network as SCL:
   "PID_Compact_2"(Setpoint := "PID_Bon4_SP",   // PID_Compact
                   Input := "TT3219_Bon4_Sim",
                   ManualEnable := "PID_Bon4_ManualEnable",
                   ManualValue := "PID_Bon4_ManualValue",
                   Reset := "PID_Bon4_Reset_Eff",
                   Output => "PID_Bon4_CV",
                   State => "PID_Bon4_State",
                   Error => "PID_Bon4_ErrorBits");
END_REGION

REGION Network 9: Detect PID Bon 4 Error
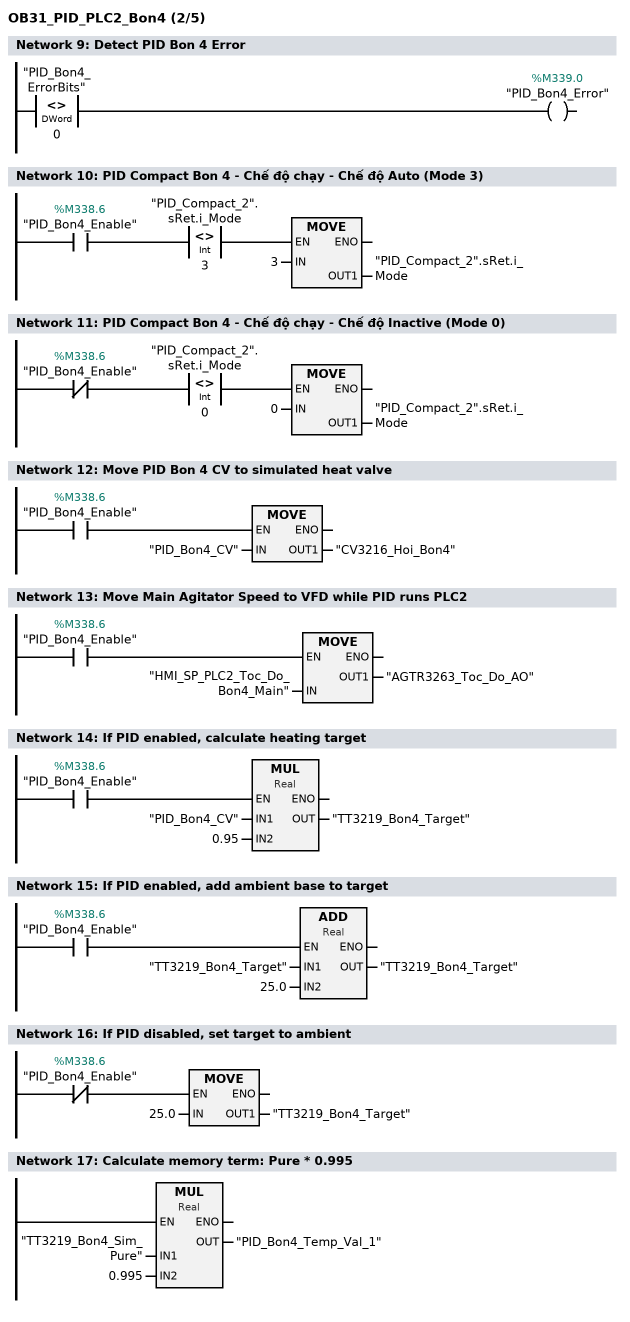
   RUNG wire#powerrail
      { S7_Templates := "SrcType := DWord" } NE_Contact(in1 := "PID_Bon4_ErrorBits", in2 := 0)
      Coil( "PID_Bon4_Error" )
   END_RUNG
   // the same network as SCL:
   "PID_Bon4_Error" := "PID_Bon4_ErrorBits" <> 0;
END_REGION

REGION Network 10: PID Compact Bon 4 - Chế độ chạy - Chế độ Auto (Mode 3)
   RUNG wire#powerrail
      Contact( "PID_Bon4_Enable" )
      { S7_Templates := "SrcType := Int" } NE_Contact(in1 := "PID_Compact_2".sRet.i_Mode, in2 := 3)
      { S7_GenerateENO := "TRUE" } Move(in := 3, out1 => "PID_Compact_2".sRet.i_Mode)
   END_RUNG
   // the same network as SCL:
   IF "PID_Bon4_Enable" AND ("PID_Compact_2".sRet.i_Mode <> 3) THEN "PID_Compact_2".sRet.i_Mode := 3; END_IF;
END_REGION

REGION Network 11: PID Compact Bon 4 - Chế độ chạy - Chế độ Inactive (Mode 0)
   RUNG wire#powerrail
      I_Contact( "PID_Bon4_Enable" )
      { S7_Templates := "SrcType := Int" } NE_Contact(in1 := "PID_Compact_2".sRet.i_Mode, in2 := 0)
      { S7_GenerateENO := "TRUE" } Move(in := 0, out1 => "PID_Compact_2".sRet.i_Mode)
   END_RUNG
   // the same network as SCL:
   IF NOT "PID_Bon4_Enable" AND ("PID_Compact_2".sRet.i_Mode <> 0) THEN
       "PID_Compact_2".sRet.i_Mode := 0;
   END_IF;
END_REGION

REGION Network 12: Move PID Bon 4 CV to simulated heat valve
   RUNG wire#powerrail
      Contact( "PID_Bon4_Enable" )
      { S7_GenerateENO := "TRUE" } Move(in := "PID_Bon4_CV", out1 => "CV3216_Hoi_Bon4")
   END_RUNG
   // the same network as SCL:
   IF "PID_Bon4_Enable" THEN "CV3216_Hoi_Bon4" := "PID_Bon4_CV"; END_IF;
END_REGION

REGION Network 13: Move Main Agitator Speed to VFD while PID runs PLC2
   RUNG wire#powerrail
      Contact( "PID_Bon4_Enable" )
      { S7_GenerateENO := "TRUE" } Move(in := "HMI_SP_PLC2_Toc_Do_Bon4_Main", out1 => "AGTR3263_Toc_Do_AO")
   END_RUNG
   // the same network as SCL:
   IF "PID_Bon4_Enable" THEN "AGTR3263_Toc_Do_AO" := "HMI_SP_PLC2_Toc_Do_Bon4_Main"; END_IF;
END_REGION

REGION Network 14: If PID enabled, calculate heating target
   RUNG wire#powerrail
      Contact( "PID_Bon4_Enable" )
      { S7_Templates := "SrcType := Real"; S7_GenerateENO := "TRUE" } Mul(in1 := "PID_Bon4_CV", in2 := 0.95, out => "TT3219_Bon4_Target")
   END_RUNG
   // the same network as SCL:
   IF "PID_Bon4_Enable" THEN "TT3219_Bon4_Target" := "PID_Bon4_CV" * 0.95; END_IF;
END_REGION

REGION Network 15: If PID enabled, add ambient base to target
   RUNG wire#powerrail
      Contact( "PID_Bon4_Enable" )
      { S7_Templates := "SrcType := Real"; S7_GenerateENO := "TRUE" } Add(in1 := "TT3219_Bon4_Target", in2 := 25.0, out => "TT3219_Bon4_Target")
   END_RUNG
   // the same network as SCL:
   IF "PID_Bon4_Enable" THEN "TT3219_Bon4_Target" := "TT3219_Bon4_Target" + 25.0; END_IF;
END_REGION

REGION Network 16: If PID disabled, set target to ambient
   RUNG wire#powerrail
      I_Contact( "PID_Bon4_Enable" )
      { S7_GenerateENO := "TRUE" } Move(in := 25.0, out1 => "TT3219_Bon4_Target")
   END_RUNG
   // the same network as SCL:
   IF NOT "PID_Bon4_Enable" THEN "TT3219_Bon4_Target" := 25.0; END_IF;
END_REGION

REGION Network 17: Calculate memory term: Pure * 0.995
   RUNG wire#powerrail
      { S7_Templates := "SrcType := Real"; S7_GenerateENO := "TRUE" } Mul(in1 := "TT3219_Bon4_Sim_Pure", in2 := 0.995, out => "PID_Bon4_Temp_Val_1")
   END_RUNG
   // the same network as SCL:
   "PID_Bon4_Temp_Val_1" := "TT3219_Bon4_Sim_Pure" * 0.995;
END_REGION

REGION Network 18: Calculate target term: Target * 0.005
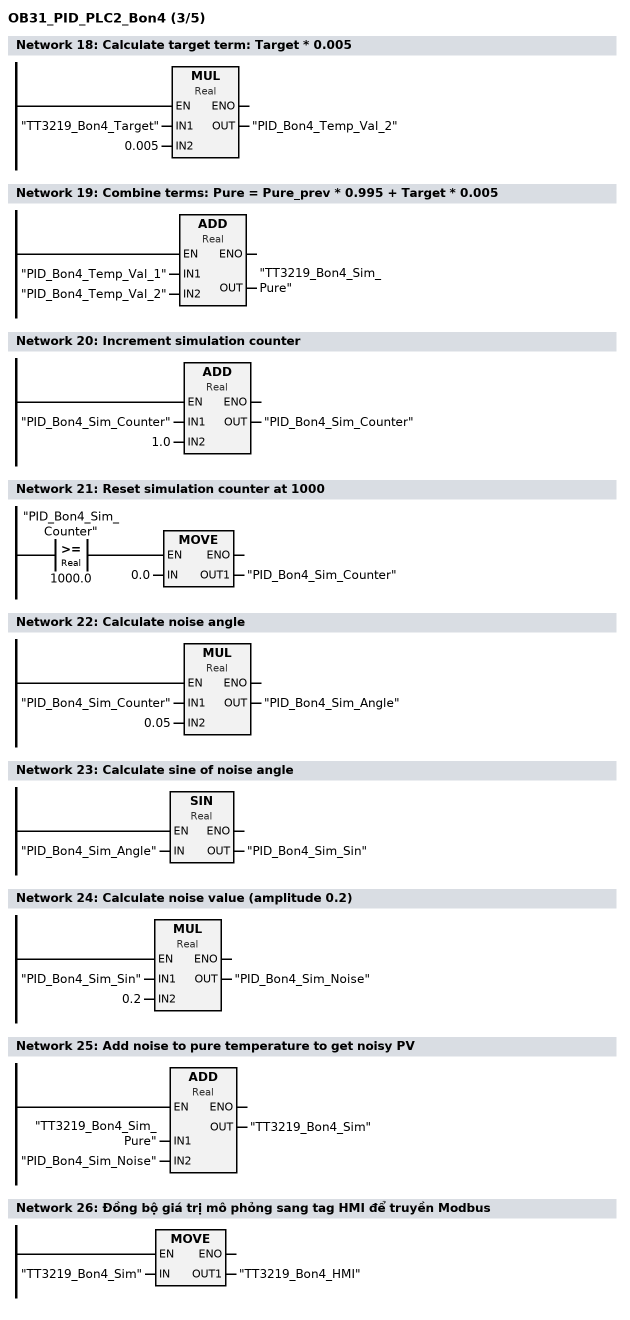
   RUNG wire#powerrail
      { S7_Templates := "SrcType := Real"; S7_GenerateENO := "TRUE" } Mul(in1 := "TT3219_Bon4_Target", in2 := 0.005, out => "PID_Bon4_Temp_Val_2")
   END_RUNG
   // the same network as SCL:
   "PID_Bon4_Temp_Val_2" := "TT3219_Bon4_Target" * 0.005;
END_REGION

REGION Network 19: Combine terms: Pure = Pure_prev * 0.995 + Target * 0.005
   RUNG wire#powerrail
      { S7_Templates := "SrcType := Real"; S7_GenerateENO := "TRUE" } Add(in1 := "PID_Bon4_Temp_Val_1", in2 := "PID_Bon4_Temp_Val_2", out => "TT3219_Bon4_Sim_Pure")
   END_RUNG
   // the same network as SCL:
   "TT3219_Bon4_Sim_Pure" := "PID_Bon4_Temp_Val_1" + "PID_Bon4_Temp_Val_2";
END_REGION

REGION Network 20: Increment simulation counter
   RUNG wire#powerrail
      { S7_Templates := "SrcType := Real"; S7_GenerateENO := "TRUE" } Add(in1 := "PID_Bon4_Sim_Counter", in2 := 1.0, out => "PID_Bon4_Sim_Counter")
   END_RUNG
   // the same network as SCL:
   "PID_Bon4_Sim_Counter" := "PID_Bon4_Sim_Counter" + 1.0;
END_REGION

REGION Network 21: Reset simulation counter at 1000
   RUNG wire#powerrail
      { S7_Templates := "SrcType := Real" } GE_Contact(in1 := "PID_Bon4_Sim_Counter", in2 := 1000.0)
      { S7_GenerateENO := "TRUE" } Move(in := 0.0, out1 => "PID_Bon4_Sim_Counter")
   END_RUNG
   // the same network as SCL:
   IF "PID_Bon4_Sim_Counter" >= 1000.0 THEN "PID_Bon4_Sim_Counter" := 0.0; END_IF;
END_REGION

REGION Network 22: Calculate noise angle
   RUNG wire#powerrail
      { S7_Templates := "SrcType := Real"; S7_GenerateENO := "TRUE" } Mul(in1 := "PID_Bon4_Sim_Counter", in2 := 0.05, out => "PID_Bon4_Sim_Angle")
   END_RUNG
   // the same network as SCL:
   "PID_Bon4_Sim_Angle" := "PID_Bon4_Sim_Counter" * 0.05;
END_REGION

REGION Network 23: Calculate sine of noise angle
   "PID_Bon4_Sim_Sin" := SIN("PID_Bon4_Sim_Angle");
END_REGION

REGION Network 24: Calculate noise value (amplitude 0.2)
   RUNG wire#powerrail
      { S7_Templates := "SrcType := Real"; S7_GenerateENO := "TRUE" } Mul(in1 := "PID_Bon4_Sim_Sin", in2 := 0.2, out => "PID_Bon4_Sim_Noise")
   END_RUNG
   // the same network as SCL:
   "PID_Bon4_Sim_Noise" := "PID_Bon4_Sim_Sin" * 0.2;
END_REGION

REGION Network 25: Add noise to pure temperature to get noisy PV
   RUNG wire#powerrail
      { S7_Templates := "SrcType := Real"; S7_GenerateENO := "TRUE" } Add(in1 := "TT3219_Bon4_Sim_Pure", in2 := "PID_Bon4_Sim_Noise", out => "TT3219_Bon4_Sim")
   END_RUNG
   // the same network as SCL:
   "TT3219_Bon4_Sim" := "TT3219_Bon4_Sim_Pure" + "PID_Bon4_Sim_Noise";
END_REGION

REGION Network 26: Đồng bộ giá trị mô phỏng sang tag HMI để truyền Modbus
   RUNG wire#powerrail
      { S7_GenerateENO := "TRUE" } Move(in := "TT3219_Bon4_Sim", out1 => "TT3219_Bon4_HMI")
   END_RUNG
   // the same network as SCL:
   "TT3219_Bon4_HMI" := "TT3219_Bon4_Sim";
END_REGION

REGION Network 27: Sim Bồn 3: Tăng FQ và LT khi dosing
